KUKA KRL data list: ps_a_ltb_geo_x01.dat

&ACCESS RVO1
&COMMENT Solda Atego LTB
&PARAM DISKPATH = KRC:\R1\Program\OLP
DEFDAT ps_a_ltb_geo_x01
;FOLD EXTERNAL DECLARATIONS;%{PE}%MKUKATPBASIS,%CEXT,%VCOMMON,%P
;FOLD GRIPPERTECH EXT
EXT  H50 (INT  :IN,INT  :IN,INT  :IN,GRP_TYP  :IN )
;ENDFOLD (GRIPPERTECH EXT)
;FOLD SPOTTECH EXT
EXT  USERSPOT (S_COMMAND  :IN,SPOT_TYPE  :IN )
;ENDFOLD (SPOTTECH EXT)
;FOLD BASISTECH EXT;%{PE}%MKUKATPBASIS,%CEXT,%VEXT,%P
EXT  BAS (BAS_COMMAND  :IN,REAL  :IN )
DECL INT SUCCESS
;ENDFOLD (BASISTECH EXT)
;FOLD USER EXT;%{E}%MKUKATPUSER,%CEXT,%VEXT,%P
;Make your modifications here

;ENDFOLD (USER EXT)
;ENDFOLD (EXTERNAL DECLARATIONS)
DECL FDAT Fl005={TOOL_NO 2,BASE_NO 3,IPO_FRAME #BASE,POINT2[] " ",TQ_STATE FALSE}
DECL PDAT PP_OLP2={VEL 100.0,ACC 100.0,APO_DIST 20.0,APO_MODE #CDIS}
DECL E6POS Xl005={X 1312.45898,Y 161.401306,Z 2358.82397,A 138.055695,B 49.2517204,C -31.9309597,S 2,T 10,E1 0.0,E2 0.0,E3 0.0,E4 0.0,E5 0.0,E6 0.0}
DECL FDAT Fl010={TOOL_NO 2,BASE_NO 3,IPO_FRAME #BASE,POINT2[] " "}
DECL PDAT PP_OLP3={VEL 100.0,ACC 100.0,APO_DIST 20.0,APO_MODE #CDIS}
DECL E6POS Xl010={X 1099.32495,Y 478.981415,Z 1743.81201,A 120.314499,B 19.6099892,C -13.0668297,S 2,T 10,E1 0.0,E2 0.0,E3 0.0,E4 0.0,E5 0.0,E6 0.0}
DECL FDAT Fl015={TOOL_NO 2,BASE_NO 3,IPO_FRAME #BASE,POINT2[] " ",TQ_STATE FALSE}
DECL E6POS Xl015={X 661.974487,Y 862.0224,Z 1485.94897,A 120.333702,B 9.80480957,C -0.70352149,S 2,T 10,E1 0.0,E2 0.0,E3 0.0,E4 0.0,E5 0.0,E6 0.0}
DECL FDAT Fl020={TOOL_NO 2,BASE_NO 3,IPO_FRAME #BASE,POINT2[] " ",TQ_STATE FALSE}
DECL PDAT PP_OLP4={VEL 100.0,ACC 100.0,APO_DIST 1.0,APO_MODE #CDIS}
DECL E6POS Xl020={X 658.155701,Y 906.481018,Z 1479.59802,A 120.333801,B 9.80491829,C -0.703368127,S 2,T 10,E1 0.0,E2 0.0,E3 0.0,E4 0.0,E5 0.0,E6 0.0}
DECL FDAT FSWP_60_9850={TOOL_NO 2,BASE_NO 3,IPO_FRAME #BASE,POINT2[] " ",TQ_STATE FALSE}
DECL E6POS XSWP_60_9850={X 650.992371,Y 922.430725,Z 1484.68604,A 120.333,B 9.8059864,C -0.703050911,S 2,T 10,E1 0.0,E2 0.0,E3 0.0,E4 0.0,E5 0.0,E6 0.0}
DECL LDAT LL_OLP2={VEL 2.0,ACC 100.0,APO_DIST 0.0,APO_FAC 0.0,ORI_TYP #VAR,CIRC_TYP #BASE,JERK_FAC 50.0}
DECL FDAT Fl025={TOOL_NO 2,BASE_NO 3,IPO_FRAME #BASE,POINT2[] " ",TQ_STATE FALSE}
DECL PDAT PP_OLP5={VEL 100.0,ACC 100.0,APO_DIST 1.0,APO_MODE #CDIS}
DECL E6POS Xl025={X 673.995117,Y 879.40979,Z 1485.01794,A 120.333801,B 9.80493546,C -0.703359783,S 2,T 10,E1 0.0,E2 0.0,E3 0.0,E4 0.0,E5 0.0,E6 0.0}
DECL FDAT Fl030={TOOL_NO 2,BASE_NO 3,IPO_FRAME #BASE,POINT2[] " "}
DECL PDAT PP_OLP6={VEL 100.0,ACC 100.0,APO_DIST 20.0,APO_MODE #CDIS}
DECL E6POS Xl030={X 679.488281,Y 831.263184,Z 1526.35303,A 120.333801,B 9.80495071,C -0.703492999,S 2,T 10,E1 0.0,E2 0.0,E3 0.0,E4 0.0,E5 0.0,E6 0.0}
DECL FDAT Fl075={TOOL_NO 2,BASE_NO 3,IPO_FRAME #BASE,POINT2[] " "}
DECL PDAT PP_OLP12={VEL 100.0,ACC 100.0,APO_DIST 10.0,APO_MODE #CDIS}
DECL E6POS Xl075={X 1053.93103,Y 888.187012,Z 1501.89294,A 110.206001,B 7.66410017,C 0.278800011,S 2,T 10}
DECL FDAT Fl080={TOOL_NO 2,BASE_NO 3,IPO_FRAME #BASE,POINT2[] " ",TQ_STATE FALSE}
DECL PDAT PP_OLP13={VEL 100.0,ACC 100.0,APO_DIST 1.0,APO_MODE #CDIS}
DECL E6POS Xl080={X 1042.37305,Y 937.541321,Z 1495.12097,A 110.206001,B 7.66410017,C 0.278799713,S 2,T 10,E1 0.0,E2 0.0,E3 0.0,E4 0.0,E5 0.0,E6 0.0}
DECL FDAT FSWP_60_9830={TOOL_NO 2,BASE_NO 3,IPO_FRAME #BASE,POINT2[] " ",TQ_STATE FALSE}
DECL E6POS XSWP_60_9830={X 1047.45996,Y 935.341187,Z 1503.255,A 105.468498,B 7.6633358,C -0.35240531,S 2,T 10,E1 0.0,E2 0.0,E3 0.0,E4 0.0,E5 0.0,E6 0.0}
DECL LDAT LL_OLP7={VEL 2.0,ACC 100.0,APO_DIST 0.0,APO_FAC 0.0,ORI_TYP #VAR,CIRC_TYP #BASE,JERK_FAC 50.0}
DECL FDAT Fl085={TOOL_NO 2,BASE_NO 3,IPO_FRAME #BASE,POINT2[] " ",TQ_STATE FALSE}
DECL PDAT PP_OLP14={VEL 100.0,ACC 100.0,APO_DIST 10.0,APO_MODE #CDIS}
DECL E6POS Xl085={X 1047.91394,Y 934.013428,Z 1492.54199,A 110.206001,B 7.66410017,C 0.278799713,S 2,T 10,E1 0.0,E2 0.0,E3 0.0,E4 0.0,E5 0.0,E6 0.0}
DECL FDAT Fl090={TOOL_NO 2,BASE_NO 3,IPO_FRAME #BASE,POINT2[] " "}
DECL PDAT PP_OLP15={VEL 100.0,ACC 100.0,APO_DIST 20.0,APO_MODE #CDIS}
DECL E6POS Xl090={X 1054.13501,Y 877.552979,Z 1496.93701,A 110.206001,B 7.66410017,C 0.278800011,S 2,T 10}
DECL FDAT Fl095={TOOL_NO 2,BASE_NO 3,IPO_FRAME #BASE,POINT2[] " "}
DECL PDAT PP_OLP16={VEL 100.0,ACC 100.0,APO_DIST 20.0,APO_MODE #CDIS}
DECL E6POS Xl095={X 1235.46899,Y 833.687683,Z 1509.99805,A 95.0815277,B 7.10638905,C -1.278669,S 2,T 10,E1 0.0,E2 0.0,E3 0.0,E4 0.0,E5 0.0,E6 0.0}
DECL FDAT Fl100={TOOL_NO 2,BASE_NO 3,IPO_FRAME #BASE,POINT2[] " "}
DECL PDAT PP_OLP17={VEL 100.0,ACC 100.0,APO_DIST 1.0,APO_MODE #CDIS}
DECL E6POS Xl100={X 1220.69995,Y 941.12323,Z 1501.41797,A 95.0815964,B 7.10640001,C -0.278800011,S 2,T 10,E1 0.0,E2 0.0,E3 0.0,E4 0.0,E5 0.0,E6 0.0}
DECL FDAT FSWP_60_9820={TOOL_NO 2,BASE_NO 3,IPO_FRAME #BASE,POINT2[] " ",TQ_STATE FALSE}
DECL E6POS XSWP_60_9820={X 1228.35999,Y 938.071594,Z 1507.35901,A 95.0815964,B 7.10639477,C -0.278758287,S 2,T 10,E1 0.0,E2 0.0,E3 0.0,E4 0.0,E5 0.0,E6 0.0}
DECL LDAT LL_OLP8={VEL 2.0,ACC 100.0,APO_DIST 0.0,APO_FAC 0.0,ORI_TYP #VAR,CIRC_TYP #BASE,JERK_FAC 50.0}
DECL FDAT Fl105={TOOL_NO 2,BASE_NO 3,IPO_FRAME #BASE,POINT2[] " ",TQ_STATE FALSE}
DECL PDAT PP_OLP18={VEL 100.0,ACC 100.0,APO_DIST 5.0,APO_MODE #CDIS}
DECL E6POS Xl105={X 1221.16797,Y 935.86438,Z 1502.07605,A 95.0815964,B 7.10640001,C -0.278800011,S 2,T 10,E1 0.0,E2 0.0,E3 0.0,E4 0.0,E5 0.0,E6 0.0}
DECL FDAT Fl110={TOOL_NO 2,BASE_NO 3,IPO_FRAME #BASE,POINT2[] " "}
DECL PDAT PP_OLP19={VEL 100.0,ACC 100.0,APO_DIST 20.0,APO_MODE #CDIS}
DECL E6POS Xl110={X 1240.21802,Y 780.291016,Z 1516.68005,A 95.0814972,B 7.10640001,C -1.27869999,S 2,T 10}
DECL FDAT Fl115={TOOL_NO 2,BASE_NO 3,IPO_FRAME #BASE,POINT2[] " "}
DECL PDAT PP_OLP20={VEL 100.0,ACC 100.0,APO_DIST 20.0,APO_MODE #CDIS}
DECL E6POS Xl115={X 1330.44897,Y 420.916992,Z 1021.96503,A 41.7639008,B 75.9056015,C 134.514694,S 2,T 10}
DECL FDAT Fl120={TOOL_NO 2,BASE_NO 3,IPO_FRAME #BASE,POINT2[] " "}
DECL PDAT PP_OLP21={VEL 100.0,ACC 100.0,APO_DIST 10.0,APO_MODE #CDIS}
DECL E6POS Xl120={X 1430.45703,Y 920.916016,Z 371.963013,A 69.623497,B 58.540699,C 160.565796,S 2,T 8}
DECL FDAT Fl125={TOOL_NO 2,BASE_NO 3,IPO_FRAME #BASE,POINT2[] " "}
DECL PDAT PP_OLP22={VEL 100.0,ACC 100.0,APO_DIST 1.0,APO_MODE #CDIS}
DECL E6POS Xl125={X 1430.50403,Y 1010.90399,Z 366.421509,A 69.6233978,B 58.540699,C 160.565704,S 2,T 8,E1 0.0,E2 0.0,E3 0.0,E4 0.0,E5 0.0,E6 0.0}
DECL FDAT Fl130={TOOL_NO 2,BASE_NO 3,IPO_FRAME #BASE,POINT2[] " ",TQ_STATE FALSE}
DECL E6POS Xl130={X 1432.80505,Y 1017.59302,Z 344.019592,A 60.8482018,B 67.7460022,C 152.708603,S 2,T 8,E1 0.0,E2 0.0,E3 0.0,E4 0.0,E5 0.0,E6 0.0}
DECL LDAT LL_OLP9={VEL 1.0,ACC 100.0,APO_DIST 1.0,APO_FAC 0.0,ORI_TYP #VAR,CIRC_TYP #BASE,JERK_FAC 50.0}
DECL FDAT Fl135={TOOL_NO 2,BASE_NO 3,IPO_FRAME #BASE,POINT2[] " "}
DECL E6POS Xl135={X 1404.30798,Y 1011.31897,Z 333.189606,A 176.413498,B 85.4335403,C -90.0502014,S 2,T 9,E1 0.0,E2 0.0,E3 0.0,E4 0.0,E5 0.0,E6 0.0}
DECL LDAT LL_OLP10={VEL 1.0,ACC 100.0,APO_DIST 1.0,APO_FAC 0.0,ORI_TYP #VAR,CIRC_TYP #BASE,JERK_FAC 50.0}
DECL FDAT FSWP_60_9556={TOOL_NO 2,BASE_NO 3,IPO_FRAME #BASE,POINT2[] " ",TQ_STATE FALSE}
DECL E6POS XSWP_60_9556={X 1399.95203,Y 1005.73297,Z 339.989105,A 176.371597,B 82.4862366,C -89.9990616,S 2,T 41,E1 0.0,E2 0.0,E3 0.0,E4 0.0,E5 0.0,E6 0.0}
DECL LDAT LL_OLP11={VEL 2.0,ACC 100.0,APO_DIST 0.0,APO_FAC 0.0,ORI_TYP #VAR,CIRC_TYP #BASE,JERK_FAC 50.0}
DECL FDAT FSWP_60_9568={TOOL_NO 2,BASE_NO 3,IPO_FRAME #BASE,POINT2[] " ",TQ_STATE FALSE}
DECL E6POS XSWP_60_9568={X 1572.35706,Y 996.624878,Z 306.298309,A -3.66327906,B 52.9997711,C 89.9598618,S 2,T 9,E1 0.0,E2 0.0,E3 0.0,E4 0.0,E5 0.0,E6 0.0}
DECL LDAT LL_OLP14={VEL 2.0,ACC 100.0,APO_DIST 0.0,APO_FAC 0.0,ORI_TYP #VAR,CIRC_TYP #BASE,JERK_FAC 50.0}
DECL FDAT Fl150={TOOL_NO 2,BASE_NO 3,IPO_FRAME #BASE,POINT2[] " ",TQ_STATE FALSE}
DECL E6POS Xl150={X 1501.948,Y 1015.54901,Z 314.006989,A 6.11479998,B 59.6772995,C 97.5519028,S 2,T 9,E1 0.0,E2 0.0,E3 0.0,E4 0.0,E5 0.0,E6 0.0}
DECL LDAT LL_OLP15={VEL 1.0,ACC 100.0,APO_DIST 5.0,APO_FAC 0.0,ORI_TYP #VAR,CIRC_TYP #BASE,JERK_FAC 50.0}
DECL FDAT Fl155={TOOL_NO 2,BASE_NO 3,IPO_FRAME #BASE,POINT2[] " "}
DECL E6POS Xl155={X 1430.505,Y 1010.64301,Z 363.86969,A 69.623497,B 58.540699,C 160.565704,S 2,T 8,E1 0.0,E2 0.0,E3 0.0,E4 0.0,E5 0.0,E6 0.0}
DECL LDAT LL_OLP16={VEL 1.0,ACC 100.0,APO_DIST 2.0,APO_FAC 0.0,ORI_TYP #VAR,CIRC_TYP #BASE,JERK_FAC 50.0}
DECL FDAT Fl160={TOOL_NO 2,BASE_NO 3,IPO_FRAME #BASE,POINT2[] " ",TQ_STATE FALSE}
DECL PDAT PP_OLP23={VEL 100.0,ACC 100.0,APO_DIST 10.0,APO_MODE #CDIS}
DECL E6POS Xl160={X 1430.45496,Y 920.916016,Z 371.963013,A 69.623497,B 58.540699,C 160.565704,S 2,T 8}
DECL FDAT Fl165={TOOL_NO 2,BASE_NO 3,IPO_FRAME #BASE,POINT2[] " "}
DECL PDAT PP_OLP24={VEL 100.0,ACC 100.0,APO_DIST 20.0,APO_MODE #CDIS}
DECL E6POS Xl165={X 2150.21997,Y 916.004028,Z 296.890991,A 90.0,B 50.0000992,C -90.0,S 2,T 41}
DECL FDAT Fl170={TOOL_NO 2,BASE_NO 3,IPO_FRAME #BASE,POINT2[] " ",TQ_STATE FALSE}
DECL E6POS Xl170={X 2210.22095,Y 936.007019,Z 296.891998,A 76.0688019,B 44.0681992,C -100.668999,S 2,T 41}
DECL LDAT LL_OLP17={VEL 1.0,ACC 100.0,APO_DIST 5.0,APO_FAC 0.0,ORI_TYP #VAR,CIRC_TYP #BASE,JERK_FAC 50.0}
DECL FDAT Fl175={TOOL_NO 2,BASE_NO 3,IPO_FRAME #BASE,POINT2[] " "}
DECL E6POS Xl175={X 2210.23511,Y 950.996521,Z 278.219299,A 90.0002594,B 50.0004005,C -89.9997406,S 2,T 41,E1 0.0,E2 0.0,E3 0.0,E4 0.0,E5 0.0,E6 0.0}
DECL LDAT LL_OLP18={VEL 1.0,ACC 100.0,APO_DIST 1.0,APO_FAC 0.0,ORI_TYP #VAR,CIRC_TYP #BASE,JERK_FAC 50.0}
DECL FDAT FSWP_60_9456={TOOL_NO 2,BASE_NO 3,IPO_FRAME #BASE,POINT2[] " ",TQ_STATE FALSE}
DECL E6POS XSWP_60_9456={X 2205.08203,Y 972.187317,Z 273.574799,A 98.7543564,B 49.6729088,C -83.3060226,S 2,T 41,E1 0.0,E2 0.0,E3 0.0,E4 0.0,E5 0.0,E6 0.0}
DECL LDAT LL_OLP19={VEL 2.0,ACC 100.0,APO_DIST 0.0,APO_FAC 0.0,ORI_TYP #VAR,CIRC_TYP #BASE,JERK_FAC 50.0}
DECL FDAT Fl180={TOOL_NO 2,BASE_NO 3,IPO_FRAME #BASE,POINT2[] " ",TQ_STATE FALSE}
DECL E6POS Xl180={X 2208.22998,Y 950.996582,Z 277.63559,A 90.000267,B 50.0004005,C -89.9997406,S 2,T 41,E1 0.0,E2 0.0,E3 0.0,E4 0.0,E5 0.0,E6 0.0}
DECL LDAT LL_OLP20={VEL 1.0,ACC 100.0,APO_DIST 5.0,APO_FAC 0.0,ORI_TYP #VAR,CIRC_TYP #BASE,JERK_FAC 50.0}
DECL FDAT Fl185={TOOL_NO 2,BASE_NO 3,IPO_FRAME #BASE,POINT2[] " "}
DECL E6POS Xl185={X 2214.52905,Y 863.063171,Z 284.3349,A 90.0,B 70.0,C -90.0,S 2,T 41,E1 0.0,E2 0.0,E3 0.0,E4 0.0,E5 0.0,E6 0.0}
DECL LDAT LL_OLP21={VEL 1.0,ACC 100.0,APO_DIST 5.0,APO_FAC 0.0,ORI_TYP #VAR,CIRC_TYP #BASE,JERK_FAC 50.0}
DECL FDAT FSWP_60_9446={TOOL_NO 2,BASE_NO 3,IPO_FRAME #BASE,POINT2[] " ",TQ_STATE FALSE}
DECL E6POS XSWP_60_9446={X 2208.25293,Y 831.700378,Z 279.504791,A 90.0002136,B 70.0000229,C -89.9997864,S 2,T 41,E1 0.0,E2 0.0,E3 0.0,E4 0.0,E5 0.0,E6 0.0}
DECL LDAT LL_OLP22={VEL 2.0,ACC 100.0,APO_DIST 0.0,APO_FAC 0.0,ORI_TYP #VAR,CIRC_TYP #BASE,JERK_FAC 50.0}
DECL FDAT Fl195={TOOL_NO 2,BASE_NO 3,IPO_FRAME #BASE,POINT2[] " "}
DECL E6POS Xl195={X 2205.21704,Y 709.570007,Z 304.463013,A 90.0,B 70.0,C -90.0,S 2,T 41}
DECL LDAT LL_OLP24={VEL 1.0,ACC 100.0,APO_DIST 5.0,APO_FAC 0.0,ORI_TYP #VAR,CIRC_TYP #BASE,JERK_FAC 50.0}
DECL FDAT Fl200={TOOL_NO 2,BASE_NO 3,IPO_FRAME #BASE,POINT2[] " "}
DECL E6POS Xl200={X 2210.23608,Y 593.166016,Z 330.933594,A 78.6753998,B 84.9012985,C -101.280998,S 2,T 9,E1 0.0,E2 0.0,E3 0.0,E4 0.0,E5 0.0,E6 0.0}
DECL LDAT LL_OLP25={VEL 1.0,ACC 100.0,APO_DIST 5.0,APO_FAC 0.0,ORI_TYP #VAR,CIRC_TYP #BASE,JERK_FAC 50.0}
DECL FDAT FSWP_60_9436={TOOL_NO 2,BASE_NO 3,IPO_FRAME #BASE,POINT2[] " ",TQ_STATE FALSE}
DECL E6POS XSWP_60_9436={X 2207.03711,Y 588.41748,Z 325.153595,A 136.424805,B 82.7309265,C -43.8064194,S 2,T 9,E1 0.0,E2 0.0,E3 0.0,E4 0.0,E5 0.0,E6 0.0}
DECL LDAT LL_OLP26={VEL 2.0,ACC 100.0,APO_DIST 0.0,APO_FAC 0.0,ORI_TYP #VAR,CIRC_TYP #BASE,JERK_FAC 50.0}
DECL FDAT Fl205={TOOL_NO 2,BASE_NO 3,IPO_FRAME #BASE,POINT2[] " ",TQ_STATE FALSE}
DECL E6POS Xl205={X 2210.21411,Y 578.169006,Z 340.212006,A 90.0,B 85.0,C -89.9999008,S 2,T 9}
DECL LDAT LL_OLP27={VEL 1.0,ACC 100.0,APO_DIST 5.0,APO_FAC 0.0,ORI_TYP #VAR,CIRC_TYP #BASE,JERK_FAC 50.0}
DECL FDAT Fl210={TOOL_NO 2,BASE_NO 3,IPO_FRAME #BASE,POINT2[] " "}
DECL E6POS Xl210={X 2205.22095,Y 478.169006,Z 460.212006,A 90.0,B 85.0,C -90.0,S 2,T 9}
DECL LDAT LL_OLP28={VEL 1.0,ACC 100.0,APO_DIST 50.0,APO_FAC 0.0,ORI_TYP #VAR,CIRC_TYP #BASE,JERK_FAC 50.0}
DECL FDAT Fl215={TOOL_NO 2,BASE_NO 3,IPO_FRAME #BASE,POINT2[] " "}
DECL E6POS Xl215={X 2212.68994,Y 350.626801,Z 477.752014,A -58.9805984,B 84.1710968,C 120.888397,S 2,T 9,E1 0.0,E2 0.0,E3 0.0,E4 0.0,E5 0.0,E6 0.0}
DECL LDAT LL_OLP29={VEL 1.0,ACC 100.0,APO_DIST 1.0,APO_FAC 0.0,ORI_TYP #VAR,CIRC_TYP #BASE,JERK_FAC 50.0}
DECL FDAT FSWP_60_9418={TOOL_NO 2,BASE_NO 3,IPO_FRAME #BASE,POINT2[] " ",TQ_STATE FALSE}
DECL E6POS XSWP_60_9418={X 2208.3291,Y 339.465393,Z 466.934204,A -153.915298,B 84.7714386,C 26.7148399,S 2,T 9,E1 0.0,E2 0.0,E3 0.0,E4 0.0,E5 0.0,E6 0.0}
DECL LDAT LL_OLP30={VEL 2.0,ACC 100.0,APO_DIST 0.0,APO_FAC 0.0,ORI_TYP #VAR,CIRC_TYP #BASE,JERK_FAC 50.0}
DECL FDAT Fl220={TOOL_NO 2,BASE_NO 3,IPO_FRAME #BASE,POINT2[] " ",TQ_STATE FALSE}
DECL E6POS Xl220={X 2210.22192,Y 329.837006,Z 477.765991,A -90.0002975,B 85.0000992,C 89.9997025,S 2,T 9}
DECL LDAT LL_OLP31={VEL 1.0,ACC 100.0,APO_DIST 5.0,APO_FAC 0.0,ORI_TYP #VAR,CIRC_TYP #BASE,JERK_FAC 50.0}
DECL FDAT Fl225={TOOL_NO 2,BASE_NO 3,IPO_FRAME #BASE,POINT2[] " "}
DECL E6POS Xl225={X 2205.26099,Y 224.826096,Z 516.190002,A -26.3003006,B 78.8312988,C 153.256699,S 2,T 9,E1 0.0,E2 0.0,E3 0.0,E4 0.0,E5 0.0,E6 0.0}
DECL LDAT LL_OLP32={VEL 1.0,ACC 100.0,APO_DIST 10.0,APO_FAC 0.0,ORI_TYP #VAR,CIRC_TYP #BASE,JERK_FAC 50.0}
DECL FDAT Fl230={TOOL_NO 2,BASE_NO 3,IPO_FRAME #BASE,POINT2[] " "}
DECL E6POS Xl230={X 2209.88208,Y 85.7576523,Z 494.679993,A -78.4449997,B 69.6200027,C 100.849403,S 2,T 9,E1 0.0,E2 0.0,E3 0.0,E4 0.0,E5 0.0,E6 0.0}
DECL LDAT LL_OLP33={VEL 1.0,ACC 100.0,APO_DIST 5.0,APO_FAC 0.0,ORI_TYP #VAR,CIRC_TYP #BASE,JERK_FAC 50.0}
DECL FDAT FSWP_60_9402={TOOL_NO 2,BASE_NO 3,IPO_FRAME #BASE,POINT2[] " ",TQ_STATE FALSE}
DECL E6POS XSWP_60_9402={X 2206.31909,Y 39.0832901,Z 481.429993,A -103.966202,B 69.3978119,C 76.3905563,S 2,T 9,E1 0.0,E2 0.0,E3 0.0,E4 0.0,E5 0.0,E6 0.0}
DECL LDAT LL_OLP34={VEL 2.0,ACC 100.0,APO_DIST 0.0,APO_FAC 0.0,ORI_TYP #VAR,CIRC_TYP #BASE,JERK_FAC 50.0}
DECL FDAT Fl235={TOOL_NO 2,BASE_NO 3,IPO_FRAME #BASE,POINT2[] " ",TQ_STATE FALSE}
DECL E6POS Xl235={X 2209.8811,Y 85.7577896,Z 502.071899,A -78.4450607,B 69.6199722,C 100.849297,S 2,T 9,E1 0.0,E2 0.0,E3 0.0,E4 0.0,E5 0.0,E6 0.0}
DECL LDAT LL_OLP35={VEL 1.0,ACC 100.0,APO_DIST 10.0,APO_FAC 0.0,ORI_TYP #VAR,CIRC_TYP #BASE,JERK_FAC 50.0}
DECL FDAT Fl240={TOOL_NO 2,BASE_NO 3,IPO_FRAME #BASE,POINT2[] " "}
DECL E6POS Xl240={X 2125.229,Y 51.7761002,Z 518.945007,A -48.5031395,B 67.3752823,C 118.888,S 2,T 9,E1 0.0,E2 0.0,E3 0.0,E4 0.0,E5 0.0,E6 0.0}
DECL LDAT LL_OLP36={VEL 1.0,ACC 100.0,APO_DIST 20.0,APO_FAC 0.0,ORI_TYP #VAR,CIRC_TYP #BASE,JERK_FAC 50.0}
DECL FDAT Fl245={TOOL_NO 2,BASE_NO 3,IPO_FRAME #BASE,POINT2[] " "}
DECL E6POS Xl245={X 2125.2229,Y -51.7659988,Z 501.994995,A 48.5036011,B 67.3753967,C -118.887802,S 2,T 40}
DECL LDAT LL_OLP37={VEL 1.0,ACC 100.0,APO_DIST 101.0,APO_FAC 0.0,ORI_TYP #VAR,CIRC_TYP #BASE,JERK_FAC 50.0}
DECL FDAT Fl250={TOOL_NO 2,BASE_NO 3,IPO_FRAME #BASE,POINT2[] " "}
DECL E6POS Xl250={X 2210.22192,Y -87.8785324,Z 501.994995,A 48.5036011,B 67.3753967,C -118.887802,S 2,T 40,E1 0.0,E2 0.0,E3 0.0,E4 0.0,E5 0.0,E6 0.0}
DECL LDAT LL_OLP38={VEL 1.0,ACC 100.0,APO_DIST 5.0,APO_FAC 0.0,ORI_TYP #VAR,CIRC_TYP #BASE,JERK_FAC 50.0}
DECL FDAT Fl255={TOOL_NO 2,BASE_NO 3,IPO_FRAME #BASE,POINT2[] " "}
DECL E6POS Xl255={X 2213.58691,Y -83.7550735,Z 486.702515,A 75.2710037,B 70.2698975,C -93.8613968,S 2,T 40,E1 0.0,E2 0.0,E3 0.0,E4 0.0,E5 0.0,E6 0.0}
DECL LDAT LL_OLP39={VEL 1.0,ACC 100.0,APO_DIST 2.0,APO_FAC 0.0,ORI_TYP #VAR,CIRC_TYP #BASE,JERK_FAC 50.0}
DECL FDAT FSWP_60_9401={TOOL_NO 2,BASE_NO 3,IPO_FRAME #BASE,POINT2[] " ",TQ_STATE FALSE}
DECL E6POS XSWP_60_9401={X 2209.38892,Y -45.844059,Z 480.638794,A 102.350197,B 69.5346603,C -77.8060226,S 2,T 40,E1 0.0,E2 0.0,E3 0.0,E4 0.0,E5 0.0,E6 0.0}
DECL LDAT LL_OLP40={VEL 2.0,ACC 100.0,APO_DIST 0.0,APO_FAC 0.0,ORI_TYP #VAR,CIRC_TYP #BASE,JERK_FAC 50.0}
DECL FDAT Fl260={TOOL_NO 2,BASE_NO 3,IPO_FRAME #BASE,POINT2[] " ",TQ_STATE FALSE}
DECL E6POS Xl260={X 2210.19409,Y -226.362305,Z 515.516724,A 26.3024998,B 78.8311005,C -153.259796,S 2,T 8,E1 0.0,E2 0.0,E3 0.0,E4 0.0,E5 0.0,E6 0.0}
DECL LDAT LL_OLP41={VEL 1.0,ACC 100.0,APO_DIST 5.0,APO_FAC 0.0,ORI_TYP #VAR,CIRC_TYP #BASE,JERK_FAC 50.0}
DECL FDAT Fl265={TOOL_NO 2,BASE_NO 3,IPO_FRAME #BASE,POINT2[] " "}
DECL E6POS Xl265={X 2211.18408,Y -349.819397,Z 475.749908,A 89.4250107,B 88.7149429,C -90.5897598,S 2,T 8,E1 0.0,E2 0.0,E3 0.0,E4 0.0,E5 0.0,E6 0.0}
DECL LDAT LL_OLP42={VEL 1.0,ACC 100.0,APO_DIST 5.0,APO_FAC 0.0,ORI_TYP #VAR,CIRC_TYP #BASE,JERK_FAC 50.0}
DECL FDAT FSWP_60_9417={TOOL_NO 2,BASE_NO 3,IPO_FRAME #BASE,POINT2[] " ",TQ_STATE FALSE}
DECL E6POS XSWP_60_9417={X 2209.16406,Y -352.611694,Z 465.538605,A 165.204895,B 84.2824936,C -14.6828499,S 2,T 8,E1 0.0,E2 0.0,E3 0.0,E4 0.0,E5 0.0,E6 0.0}
DECL LDAT LL_OLP43={VEL 2.0,ACC 100.0,APO_DIST 0.0,APO_FAC 0.0,ORI_TYP #VAR,CIRC_TYP #BASE,JERK_FAC 50.0}
DECL FDAT Fl270={TOOL_NO 2,BASE_NO 3,IPO_FRAME #BASE,POINT2[] " ",TQ_STATE FALSE}
DECL E6POS Xl270={X 2205.22095,Y -478.169006,Z 460.212006,A -90.0,B 85.0,C 90.0,S 2,T 8}
DECL LDAT LL_OLP44={VEL 1.0,ACC 100.0,APO_DIST 5.0,APO_FAC 0.0,ORI_TYP #VAR,CIRC_TYP #BASE,JERK_FAC 50.0}
DECL FDAT FSWP_60_9435={TOOL_NO 2,BASE_NO 3,IPO_FRAME #BASE,POINT2[] " ",TQ_STATE FALSE}
DECL E6POS XSWP_60_9435={X 2206.49805,Y -596.194885,Z 325.749603,A -126.132797,B 83.7971497,C 53.8362885,S 2,T 8,E1 0.0,E2 0.0,E3 0.0,E4 0.0,E5 0.0,E6 0.0}
DECL LDAT LL_OLP45={VEL 2.0,ACC 100.0,APO_DIST 0.0,APO_FAC 0.0,ORI_TYP #VAR,CIRC_TYP #BASE,JERK_FAC 50.0}
DECL FDAT Fl275={TOOL_NO 2,BASE_NO 3,IPO_FRAME #BASE,POINT2[] " ",TQ_STATE FALSE}
DECL E6POS Xl275={X 2205.21704,Y -709.570007,Z 304.463013,A -90.0,B 70.0,C 90.0,S 2,T 8}
DECL LDAT LL_OLP46={VEL 1.0,ACC 100.0,APO_DIST 5.0,APO_FAC 0.0,ORI_TYP #VAR,CIRC_TYP #BASE,JERK_FAC 50.0}
DECL FDAT FSWP_60_9445={TOOL_NO 2,BASE_NO 3,IPO_FRAME #BASE,POINT2[] " ",TQ_STATE FALSE}
DECL E6POS XSWP_60_9445={X 2207.60107,Y -835.695984,Z 272.809509,A -99.4904099,B 69.7042694,C 80.2663193,S 2,T 8,E1 0.0,E2 0.0,E3 0.0,E4 0.0,E5 0.0,E6 0.0}
DECL LDAT LL_OLP47={VEL 2.0,ACC 100.0,APO_DIST 0.0,APO_FAC 0.0,ORI_TYP #VAR,CIRC_TYP #BASE,JERK_FAC 50.0}
DECL FDAT Fl280={TOOL_NO 2,BASE_NO 3,IPO_FRAME #BASE,POINT2[] " ",TQ_STATE FALSE}
DECL E6POS Xl280={X 2205.229,Y -921.711975,Z 294.875,A -90.0,B 50.0000992,C 90.0,S 2,T 8}
DECL LDAT LL_OLP48={VEL 1.0,ACC 100.0,APO_DIST 5.0,APO_FAC 0.0,ORI_TYP #VAR,CIRC_TYP #BASE,JERK_FAC 50.0}
DECL FDAT FSWP_60_9455={TOOL_NO 2,BASE_NO 3,IPO_FRAME #BASE,POINT2[] " ",TQ_STATE FALSE}
DECL E6POS XSWP_60_9455={X 2203.65405,Y -981.330994,Z 273.67099,A -91.5469894,B 49.9690704,C 87.3450394,S 2,T 8,E1 0.0,E2 0.0,E3 0.0,E4 0.0,E5 0.0,E6 0.0}
DECL LDAT LL_OLP49={VEL 2.0,ACC 100.0,APO_DIST 0.0,APO_FAC 0.0,ORI_TYP #VAR,CIRC_TYP #BASE,JERK_FAC 50.0}
DECL FDAT Fl285={TOOL_NO 2,BASE_NO 3,IPO_FRAME #BASE,POINT2[] " ",TQ_STATE FALSE}
DECL E6POS Xl285={X 2205.26904,Y -951.011414,Z 283.177307,A -90.0000916,B 50.0001907,C 89.9999619,S 2,T 8,E1 0.0,E2 0.0,E3 0.0,E4 0.0,E5 0.0,E6 0.0}
DECL LDAT LL_OLP50={VEL 1.0,ACC 100.0,APO_DIST 2.0,APO_FAC 0.0,ORI_TYP #VAR,CIRC_TYP #BASE,JERK_FAC 50.0}
DECL FDAT Fl290={TOOL_NO 2,BASE_NO 3,IPO_FRAME #BASE,POINT2[] " "}
DECL E6POS Xl290={X 2210.24194,Y -936.011597,Z 302.306213,A -74.660202,B 48.9735985,C 101.692101,S 2,T 8,E1 0.0,E2 0.0,E3 0.0,E4 0.0,E5 0.0,E6 0.0}
DECL LDAT LL_OLP51={VEL 1.0,ACC 100.0,APO_DIST 5.0,APO_FAC 0.0,ORI_TYP #VAR,CIRC_TYP #BASE,JERK_FAC 50.0}
DECL FDAT Fl295={TOOL_NO 2,BASE_NO 3,IPO_FRAME #BASE,POINT2[] " "}
DECL E6POS Xl295={X 2150.30005,Y -916.025818,Z 317.780914,A -89.9999924,B 50.0000992,C 90.0,S 2,T 8,E1 0.0,E2 0.0,E3 0.0,E4 0.0,E5 0.0,E6 0.0}
DECL LDAT LL_OLP52={VEL 1.0,ACC 100.0,APO_DIST 20.0,APO_FAC 0.0,ORI_TYP #VAR,CIRC_TYP #BASE,JERK_FAC 50.0}
DECL FDAT Fl300={TOOL_NO 2,BASE_NO 3,IPO_FRAME #BASE,POINT2[] " ",TQ_STATE FALSE}
DECL PDAT PP_OLP25={VEL 100.0,ACC 100.0,APO_DIST 20.0,APO_MODE #CDIS}
DECL E6POS Xl300={X 1430.48596,Y -920.923828,Z 380.326599,A -69.623497,B 58.5407104,C -160.565704,S 2,T 9,E1 0.0,E2 0.0,E3 0.0,E4 0.0,E5 0.0,E6 0.0}
DECL FDAT Fl305={TOOL_NO 2,BASE_NO 3,IPO_FRAME #BASE,POINT2[] " "}
DECL PDAT PP_OLP26={VEL 100.0,ACC 100.0,APO_DIST 5.0,APO_MODE #CDIS}
DECL E6POS Xl305={X 1430.49695,Y -1010.92603,Z 364.68219,A -69.6234894,B 58.5407104,C -160.565704,S 2,T 9,E1 0.0,E2 0.0,E3 0.0,E4 0.0,E5 0.0,E6 0.0}
DECL FDAT Fl310={TOOL_NO 2,BASE_NO 3,IPO_FRAME #BASE,POINT2[] " ",TQ_STATE FALSE}
DECL E6POS Xl310={X 1504.45801,Y -1015.81799,Z 309.69101,A -6.11479998,B 59.6772995,C -97.5519028,S 2,T 40}
DECL LDAT LL_OLP53={VEL 1.0,ACC 100.0,APO_DIST 2.0,APO_FAC 0.0,ORI_TYP #VAR,CIRC_TYP #BASE,JERK_FAC 50.0}
DECL FDAT Fl315={TOOL_NO 2,BASE_NO 3,IPO_FRAME #BASE,POINT2[] " "}
DECL E6POS Xl315={X 1559.32104,Y -1000.73297,Z 296.967987,A 3.66630006,B 55.0000992,C -89.9583969,S 2,T 40}
DECL LDAT LL_OLP54={VEL 1.0,ACC 100.0,APO_DIST 2.0,APO_FAC 0.0,ORI_TYP #VAR,CIRC_TYP #BASE,JERK_FAC 50.0}
DECL FDAT FSWP_60_9567={TOOL_NO 2,BASE_NO 3,IPO_FRAME #BASE,POINT2[] " ",TQ_STATE FALSE}
DECL E6POS XSWP_60_9567={X 1561.53894,Y -999.303223,Z 297.026215,A 3.66697097,B 55.0008392,C -89.9575882,S 2,T 40,E1 0.0,E2 0.0,E3 0.0,E4 0.0,E5 0.0,E6 0.0}
DECL LDAT LL_OLP55={VEL 2.0,ACC 100.0,APO_DIST 0.0,APO_FAC 0.0,ORI_TYP #VAR,CIRC_TYP #BASE,JERK_FAC 50.0}
DECL FDAT FSWP_60_9555={TOOL_NO 2,BASE_NO 3,IPO_FRAME #BASE,POINT2[] " ",TQ_STATE FALSE}
DECL E6POS XSWP_60_9555={X 1399.047,Y -1007.28302,Z 333.780914,A -176.405594,B 80.0015793,C 89.9643173,S 2,T 8,E1 0.0,E2 0.0,E3 0.0,E4 0.0,E5 0.0,E6 0.0}
DECL LDAT LL_OLP57={VEL 2.0,ACC 100.0,APO_DIST 0.0,APO_FAC 0.0,ORI_TYP #VAR,CIRC_TYP #BASE,JERK_FAC 50.0}
DECL FDAT Fl325={TOOL_NO 2,BASE_NO 3,IPO_FRAME #BASE,POINT2[] " ",TQ_STATE FALSE}
DECL E6POS Xl325={X 1408.64404,Y -1022.89801,Z 347.390106,A -119.316399,B 72.0361023,C 145.7341,S 2,T 8,E1 0.0,E2 0.0,E3 0.0,E4 0.0,E5 0.0,E6 0.0}
DECL LDAT LL_OLP58={VEL 1.0,ACC 100.0,APO_DIST 5.0,APO_FAC 0.0,ORI_TYP #VAR,CIRC_TYP #BASE,JERK_FAC 50.0}
DECL FDAT Fl330={TOOL_NO 2,BASE_NO 3,IPO_FRAME #BASE,POINT2[] " "}
DECL E6POS Xl330={X 1430.49805,Y -1010.927,Z 364.586212,A -69.6234894,B 58.5407104,C -160.565796,S 2,T 9,E1 0.0,E2 0.0,E3 0.0,E4 0.0,E5 0.0,E6 0.0}
DECL LDAT LL_OLP59={VEL 1.0,ACC 100.0,APO_DIST 5.0,APO_FAC 0.0,ORI_TYP #VAR,CIRC_TYP #BASE,JERK_FAC 50.0}
DECL FDAT Fl335={TOOL_NO 2,BASE_NO 3,IPO_FRAME #BASE,POINT2[] " "}
DECL E6POS Xl335={X 1430.45801,Y -920.916016,Z 371.963013,A -41.7638016,B 75.9057007,C -134.514694,S 2,T 40}
DECL LDAT LL_OLP60={VEL 1.0,ACC 100.0,APO_DIST 20.0,APO_FAC 0.0,ORI_TYP #VAR,CIRC_TYP #BASE,JERK_FAC 50.0}
DECL FDAT Fl340={TOOL_NO 2,BASE_NO 3,IPO_FRAME #BASE,POINT2[] " ",TQ_STATE FALSE}
DECL PDAT PP_OLP27={VEL 100.0,ACC 100.0,APO_DIST 50.0,APO_MODE #CDIS}
DECL E6POS Xl340={X 1023.37201,Y 195.498001,Z 1177.24402,A -56.0586014,B 67.5304031,C -3.93070006,S 2,T 10}
DECL FDAT Fl345={TOOL_NO 2,BASE_NO 3,IPO_FRAME #BASE,POINT2[] " "}
DECL PDAT PP_OLP28={VEL 100.0,ACC 100.0,APO_DIST 20.0,APO_MODE #CDIS}
DECL E6POS Xl345={X 1231.26501,Y -831.768921,Z 1504.36499,A -95.0813599,B 7.10645723,C 1.27910495,S 6,T 27,E1 0.0,E2 0.0,E3 0.0,E4 0.0,E5 0.0,E6 0.0}
DECL FDAT Fl350={TOOL_NO 2,BASE_NO 3,IPO_FRAME #BASE,POINT2[] " "}
DECL PDAT PP_OLP29={VEL 100.0,ACC 100.0,APO_DIST 2.0,APO_MODE #CDIS}
DECL E6POS Xl350={X 1229.13696,Y -941.847778,Z 1502.84204,A -95.9412231,B 4.54855013,C -6.22060919,S 6,T 27,E1 0.0,E2 0.0,E3 0.0,E4 0.0,E5 0.0,E6 0.0}
DECL FDAT FSWP_60_9819={TOOL_NO 2,BASE_NO 3,IPO_FRAME #BASE,POINT2[] " ",TQ_STATE FALSE}
DECL E6POS XSWP_60_9819={X 1222.802,Y -950.658203,Z 1506.07397,A -95.8159866,B 4.79627705,C 1.52473104,S 6,T 27,E1 0.0,E2 0.0,E3 0.0,E4 0.0,E5 0.0,E6 0.0}
DECL LDAT LL_OLP61={VEL 2.0,ACC 100.0,APO_DIST 0.0,APO_FAC 0.0,ORI_TYP #VAR,CIRC_TYP #BASE,JERK_FAC 50.0}
DECL FDAT Fl355={TOOL_NO 2,BASE_NO 3,IPO_FRAME #BASE,POINT2[] " ",TQ_STATE FALSE}
DECL PDAT PP_OLP30={VEL 100.0,ACC 100.0,APO_DIST 5.0,APO_MODE #CDIS}
DECL E6POS Xl355={X 1229.13696,Y -941.846985,Z 1502.84094,A -95.9412003,B 4.5486021,C -6.22065115,S 6,T 27,E1 0.0,E2 0.0,E3 0.0,E4 0.0,E5 0.0,E6 0.0}
DECL FDAT Fl360={TOOL_NO 2,BASE_NO 3,IPO_FRAME #BASE,POINT2[] " "}
DECL PDAT PP_OLP31={VEL 100.0,ACC 100.0,APO_DIST 10.0,APO_MODE #CDIS}
DECL E6POS Xl360={X 1245.23401,Y -831.894775,Z 1502.57397,A -95.0814972,B 7.10640001,C 1.27869999,S 6,T 27,E1 0.0,E2 0.0,E3 0.0,E4 0.0,E5 0.0,E6 0.0}
DECL FDAT Fl365={TOOL_NO 2,BASE_NO 3,IPO_FRAME #BASE,POINT2[] " ",TQ_STATE FALSE}
DECL PDAT PP_OLP32={VEL 100.0,ACC 100.0,APO_DIST 10.0,APO_MODE #CDIS}
DECL E6POS Xl365={X 1054.13501,Y -877.552979,Z 1496.93701,A -110.206001,B 7.66410017,C -0.278800011,S 6,T 27}
DECL FDAT Fl370={TOOL_NO 2,BASE_NO 3,IPO_FRAME #BASE,POINT2[] " "}
DECL PDAT PP_OLP33={VEL 100.0,ACC 100.0,APO_DIST 5.0,APO_MODE #CDIS}
DECL E6POS Xl370={X 1041.78296,Y -941.79248,Z 1494.52405,A -110.206001,B 7.66410017,C -0.278800011,S 6,T 27,E1 0.0,E2 0.0,E3 0.0,E4 0.0,E5 0.0,E6 0.0}
DECL FDAT FSWP_60_9829={TOOL_NO 2,BASE_NO 3,IPO_FRAME #BASE,POINT2[] " ",TQ_STATE FALSE}
DECL E6POS XSWP_60_9829={X 1048.76794,Y -952.477783,Z 1499.80103,A -110.206299,B 7.66383219,C -0.278844714,S 6,T 26,E1 0.0,E2 0.0,E3 0.0,E4 0.0,E5 0.0,E6 0.0}
DECL LDAT LL_OLP62={VEL 2.0,ACC 100.0,APO_DIST 0.0,APO_FAC 0.0,ORI_TYP #VAR,CIRC_TYP #BASE,JERK_FAC 50.0}
DECL FDAT Fl375={TOOL_NO 2,BASE_NO 3,IPO_FRAME #BASE,POINT2[] " ",TQ_STATE FALSE}
DECL PDAT PP_OLP34={VEL 100.0,ACC 100.0,APO_DIST 10.0,APO_MODE #CDIS}
DECL E6POS Xl375={X 1064.71106,Y -879.495422,Z 1503.45703,A -110.206001,B 7.66410017,C -0.278800011,S 6,T 27,E1 0.0,E2 0.0,E3 0.0,E4 0.0,E5 0.0,E6 0.0}
DECL FDAT Fl380={TOOL_NO 2,BASE_NO 3,IPO_FRAME #BASE,POINT2[] " "}
DECL PDAT PP_OLP35={VEL 100.0,ACC 100.0,APO_DIST 10.0,APO_MODE #CDIS}
DECL E6POS Xl380={X 1070.62,Y -843.634094,Z 1565.01404,A -110.206001,B 7.66410208,C -0.278800696,S 6,T 27,E1 0.0,E2 0.0,E3 0.0,E4 0.0,E5 0.0,E6 0.0}
DECL FDAT Fl385={TOOL_NO 2,BASE_NO 3,IPO_FRAME #BASE,POINT2[] " "}
DECL PDAT PP_OLP36={VEL 100.0,ACC 100.0,APO_DIST 20.0,APO_MODE #CDIS}
DECL E6POS Xl385={X 910.014587,Y -845.905884,Z 1559.67297,A -110.206001,B 7.66410398,C -0.278801888,S 6,T 27,E1 0.0,E2 0.0,E3 0.0,E4 0.0,E5 0.0,E6 0.0}
DECL FDAT Fl420={TOOL_NO 2,BASE_NO 3,IPO_FRAME #BASE,POINT2[] " "}
DECL PDAT PP_OLP40={VEL 100.0,ACC 100.0,APO_DIST 20.0,APO_MODE #CDIS}
DECL E6POS Xl420={X 660.002075,Y -860.751282,Z 1542.66504,A -120.333801,B 9.80494022,C 0.703443885,S 6,T 58,E1 0.0,E2 0.0,E3 0.0,E4 0.0,E5 0.0,E6 0.0}
DECL FDAT Fl425={TOOL_NO 2,BASE_NO 3,IPO_FRAME #BASE,POINT2[] " ",TQ_STATE FALSE}
DECL PDAT PP_OLP41={VEL 100.0,ACC 100.0,APO_DIST 10.0,APO_MODE #CDIS}
DECL E6POS Xl425={X 646.763,Y -884.752014,Z 1480.66895,A -120.333801,B 9.80490017,C 0.703499973,S 6,T 58}
DECL FDAT Fl430={TOOL_NO 2,BASE_NO 3,IPO_FRAME #BASE,POINT2[] " "}
DECL PDAT PP_OLP42={VEL 100.0,ACC 100.0,APO_DIST 2.0,APO_MODE #CDIS}
DECL E6POS Xl430={X 632.411377,Y -939.182617,Z 1471.48401,A -120.333801,B 9.80489922,C 0.703500926,S 6,T 58,E1 0.0,E2 0.0,E3 0.0,E4 0.0,E5 0.0,E6 0.0}
DECL FDAT FSWP_60_9849={TOOL_NO 2,BASE_NO 3,IPO_FRAME #BASE,POINT2[] " ",TQ_STATE FALSE}
DECL E6POS XSWP_60_9849={X 648.606018,Y -944.173279,Z 1474.62,A -110.055496,B 9.46926117,C 2.36206508,S 6,T 58,E1 0.0,E2 0.0,E3 0.0,E4 0.0,E5 0.0,E6 0.0}
DECL LDAT LL_OLP67={VEL 2.0,ACC 100.0,APO_DIST 0.0,APO_FAC 0.0,ORI_TYP #VAR,CIRC_TYP #BASE,JERK_FAC 50.0}
DECL FDAT Fl435={TOOL_NO 2,BASE_NO 3,IPO_FRAME #BASE,POINT2[] " ",TQ_STATE FALSE}
DECL E6POS Xl435={X 632.411377,Y -939.182617,Z 1471.48401,A -120.333801,B 9.80489922,C 0.703500926,S 6,T 58,E1 0.0,E2 0.0,E3 0.0,E4 0.0,E5 0.0,E6 0.0}
DECL FDAT Fl440={TOOL_NO 2,BASE_NO 3,IPO_FRAME #BASE,POINT2[] " "}
DECL PDAT PP_OLP44={VEL 100.0,ACC 100.0,APO_DIST 10.0,APO_MODE #CDIS}
DECL E6POS Xl440={X 646.763977,Y -884.752014,Z 1480.66895,A -120.333801,B 9.80490017,C 0.703499973,S 6,T 58}
DECL FDAT Fl445={TOOL_NO 2,BASE_NO 3,IPO_FRAME #BASE,POINT2[] " ",TQ_STATE FALSE}
DECL E6POS Xl445={X 903.630981,Y -565.390015,Z 1544.61304,A -115.101402,B 14.6844997,C 2.03340006,S 6,T 27}
DECL LDAT LL_OLP68={VEL 1.0,ACC 100.0,APO_DIST 50.0,APO_FAC 0.0,ORI_TYP #VAR,CIRC_TYP #BASE,JERK_FAC 50.0}
DECL FDAT Fl450={TOOL_NO 2,BASE_NO 3,IPO_FRAME #BASE,POINT2[] " ",TQ_STATE FALSE}
DECL PDAT PP_OLP45={VEL 100.0,ACC 100.0,APO_DIST 50.0,APO_MODE #CDIS}
DECL E6POS Xl450={X 1399.95703,Y -542.234924,Z 2580.37402,A -75.9914017,B 22.5326004,C -25.0158005,S 6,T 27,E1 0.0,E2 0.0,E3 0.0,E4 0.0,E5 0.0,E6 0.0}
DECL BASIS_SUGG_T LAST_BASIS={POINT1[] "P0                      ",POINT2[] "P0                      ",CP_PARAMS[] "CPDAT0                  ",PTP_PARAMS[] "PDAT0                   ",CONT[] "                        ",CP_VEL[] "2.0                     ",PTP_VEL[] " 100                    ",SYNC_PARAMS[] "SYNCDAT                 ",SPL_NAME[] "S0                      "}
DECL PDAT PP_OLP47={VEL 100.0,ACC 100.0,APO_DIST 50.0,APO_MODE #CDIS}
DECL E6POS Xl006={X 1052.75195,Y 58.7190018,Z 2073.41504,A -29.1716995,B 74.7963028,C -24.9258003,S 2,T 3}
DECL FDAT Fl006={TOOL_NO 2,BASE_NO 3,IPO_FRAME #BASE,POINT2[] " ",TQ_STATE FALSE}
DECL PDAT PP_OLP48={VEL 100.0,ACC 100.0,APO_DIST 0.0}
DECL E6POS Xl011={X 788.399475,Y 515.901306,Z 807.937988,A -165.150803,B 79.6066818,C -105.500198,S 2,T 8,E1 0.0,E2 0.0,E3 0.0,E4 0.0,E5 0.0,E6 0.0}
DECL FDAT Fl011={TOOL_NO 2,BASE_NO 3,IPO_FRAME #BASE,POINT2[] " ",TQ_STATE FALSE}
DECL LDAT LL_OLP69={VEL 2.0,ACC 100.0,APO_DIST 50.0,APO_FAC 0.0,ORI_TYP #VAR,CIRC_TYP #BASE,JERK_FAC 50.0}
DECL E6POS Xl016={X 293.170685,Y 908.471497,Z -4.25657701,A -179.468506,B 64.3328323,C -98.5837173,S 2,T 41,E1 0.0,E2 0.0,E3 0.0,E4 0.0,E5 0.0,E6 0.0}
DECL FDAT Fl016={TOOL_NO 2,BASE_NO 3,IPO_FRAME #BASE,POINT2[] " ",TQ_STATE FALSE}
DECL LDAT LL_OLP70={VEL 1.0,ACC 100.0,APO_DIST 50.0,APO_FAC 0.0,ORI_TYP #VAR,CIRC_TYP #BASE,JERK_FAC 50.0}
DECL E6POS Xl021={X 247.672897,Y 971.730774,Z -5.53645706,A -178.005096,B 59.3805809,C -97.2920685,S 2,T 41,E1 0.0,E2 0.0,E3 0.0,E4 0.0,E5 0.0,E6 0.0}
DECL FDAT Fl021={TOOL_NO 2,BASE_NO 3,IPO_FRAME #BASE,POINT2[] " ",TQ_STATE FALSE}
DECL LDAT LL_OLP71={VEL 1.0,ACC 100.0,APO_DIST 50.0,APO_FAC 0.0,ORI_TYP #VAR,CIRC_TYP #BASE,JERK_FAC 50.0}
DECL E6POS Xl026={X 233.621597,Y 967.395508,Z -22.1104393,A -168.154404,B 59.6471596,C -98.7977829,S 2,T 41,E1 0.0,E2 0.0,E3 0.0,E4 0.0,E5 0.0,E6 0.0}
DECL FDAT Fl026={TOOL_NO 2,BASE_NO 3,IPO_FRAME #BASE,POINT2[] " "}
DECL LDAT LL_OLP72={VEL 2.0,ACC 100.0,APO_DIST 0.0,APO_FAC 0.0,ORI_TYP #VAR,CIRC_TYP #BASE,JERK_FAC 50.0}
DECL E6POS XSWP_60_7094={X 221.0009,Y 949.254211,Z -5.67251396,A -158.217896,B 60.0425797,C -90.2032166,S 2,T 41,E1 0.0,E2 0.0,E3 0.0,E4 0.0,E5 0.0,E6 0.0}
DECL FDAT FSWP_60_7094={TOOL_NO 2,BASE_NO 3,IPO_FRAME #BASE,POINT2[] " ",TQ_STATE FALSE}
DECL LDAT LL_OLP73={VEL 2.0,ACC 100.0,APO_DIST 0.0,APO_FAC 0.0,ORI_TYP #VAR,CIRC_TYP #BASE,JERK_FAC 50.0}
DECL E6POS XSWP_60_7092={X 228.085007,Y 955.866516,Z -30.4384708,A -158.172897,B 60.0435295,C -90.218132,S 2,T 41,E1 0.0,E2 0.0,E3 0.0,E4 0.0,E5 0.0,E6 0.0}
DECL FDAT FSWP_60_7092={TOOL_NO 2,BASE_NO 3,IPO_FRAME #BASE,POINT2[] " ",TQ_STATE FALSE}
DECL LDAT LL_OLP74={VEL 2.0,ACC 100.0,APO_DIST 0.0,APO_FAC 0.0,ORI_TYP #VAR,CIRC_TYP #BASE,JERK_FAC 50.0}
DECL E6POS XSWP_60_7090={X 257.39801,Y 968.361877,Z -36.2215195,A -159.207306,B 74.1114807,C -91.3095169,S 2,T 9,E1 0.0,E2 0.0,E3 0.0,E4 0.0,E5 0.0,E6 0.0}
DECL FDAT FSWP_60_7090={TOOL_NO 2,BASE_NO 3,IPO_FRAME #BASE,POINT2[] " ",TQ_STATE FALSE}
DECL LDAT LL_OLP75={VEL 1.0,ACC 100.0,APO_DIST 50.0,APO_FAC 0.0,ORI_TYP #VAR,CIRC_TYP #BASE,JERK_FAC 50.0}
DECL E6POS Xl031={X 272.755188,Y 979.568115,Z -35.2234383,A -159.434296,B 79.5372467,C -93.4828186,S 2,T 9,E1 0.0,E2 0.0,E3 0.0,E4 0.0,E5 0.0,E6 0.0}
DECL FDAT Fl031={TOOL_NO 2,BASE_NO 3,IPO_FRAME #BASE,POINT2[] " ",TQ_STATE FALSE}
DECL LDAT LL_OLP76={VEL 2.0,ACC 100.0,APO_DIST 0.0,APO_FAC 0.0,ORI_TYP #VAR,CIRC_TYP #BASE,JERK_FAC 50.0}
DECL E6POS XSWP_60_7088={X 285.440308,Y 980.615906,Z -43.8656693,A -157.531998,B 82.9950027,C -93.2140198,S 2,T 9,E1 0.0,E2 0.0,E3 0.0,E4 0.0,E5 0.0,E6 0.0}
DECL FDAT FSWP_60_7088={TOOL_NO 2,BASE_NO 3,IPO_FRAME #BASE,POINT2[] " ",TQ_STATE FALSE}
DECL LDAT LL_OLP77={VEL 1.0,ACC 100.0,APO_DIST 50.0,APO_FAC 0.0,ORI_TYP #VAR,CIRC_TYP #BASE,JERK_FAC 50.0}
DECL E6POS Xl036={X 275.141998,Y 983.413818,Z -33.1203995,A 114.270798,B 82.9114609,C 178.523804,S 2,T 9,E1 0.0,E2 0.0,E3 0.0,E4 0.0,E5 0.0,E6 0.0}
DECL FDAT Fl036={TOOL_NO 2,BASE_NO 3,IPO_FRAME #BASE,POINT2[] " ",TQ_STATE FALSE}
DECL LDAT LL_OLP78={VEL 1.0,ACC 100.0,APO_DIST 0.0,APO_FAC 0.0,ORI_TYP #VAR,CIRC_TYP #BASE,JERK_FAC 50.0}
DECL E6POS Xl041={X 252.249496,Y 973.365784,Z -13.6638203,A -178.005096,B 59.3806686,C -97.2922668,S 2,T 41,E1 0.0,E2 0.0,E3 0.0,E4 0.0,E5 0.0,E6 0.0}
DECL FDAT Fl041={TOOL_NO 2,BASE_NO 3,IPO_FRAME #BASE,POINT2[] " "}
DECL LDAT LL_OLP79={VEL 1.0,ACC 100.0,APO_DIST 50.0,APO_FAC 0.0,ORI_TYP #VAR,CIRC_TYP #BASE,JERK_FAC 50.0}
DECL E6POS Xl046={X 295.162598,Y 908.491699,Z -0.105315603,A -179.480606,B 64.3333435,C -98.5977707,S 2,T 41,E1 0.0,E2 0.0,E3 0.0,E4 0.0,E5 0.0,E6 0.0}
DECL FDAT Fl046={TOOL_NO 2,BASE_NO 3,IPO_FRAME #BASE,POINT2[] " "}
DECL PDAT PP_OLP49={VEL 100.0,ACC 100.0,APO_DIST 50.0,APO_MODE #CDIS}
DECL E6POS Xl007={X 640.695679,Y -18.6962795,Z 885.305176,A -143.177597,B 82.1491623,C -143.1194,S 2,T 3,E1 0.0,E2 0.0,E3 0.0,E4 0.0,E5 0.0,E6 0.0}
DECL FDAT Fl007={TOOL_NO 2,BASE_NO 3,IPO_FRAME #BASE,POINT2[] " ",TQ_STATE FALSE}
DECL LDAT LL_OLP82={VEL 2.0,ACC 100.0,APO_DIST 0.0,APO_FAC 0.0,ORI_TYP #VAR,CIRC_TYP #BASE,JERK_FAC 50.0}
DECL E6POS XSWP_60_9560={X 1456.59705,Y 1001.547,Z 327.245514,A -3.69719601,B 74.9993362,C 89.9265213,S 2,T 9,E1 0.0,E2 0.0,E3 0.0,E4 0.0,E5 0.0,E6 0.0}
DECL FDAT FSWP_60_9560={TOOL_NO 2,BASE_NO 3,IPO_FRAME #BASE,POINT2[] " ",TQ_STATE FALSE}
DECL LDAT LL_OLP83={VEL 2.0,ACC 100.0,APO_DIST 0.0,APO_FAC 0.0,ORI_TYP #VAR,CIRC_TYP #BASE,JERK_FAC 50.0}
DECL E6POS XSWP_60_9564={X 1516.00195,Y 996.921692,Z 312.947388,A -3.67799711,B 67.0000992,C 89.9478989,S 2,T 9,E1 0.0,E2 0.0,E3 0.0,E4 0.0,E5 0.0,E6 0.0}
DECL FDAT FSWP_60_9564={TOOL_NO 2,BASE_NO 3,IPO_FRAME #BASE,POINT2[] " ",TQ_STATE FALSE}
DECL LDAT LL_OLP84={VEL 2.0,ACC 100.0,APO_DIST 0.0,APO_FAC 0.0,ORI_TYP #VAR,CIRC_TYP #BASE,JERK_FAC 50.0}
DECL E6POS XSWP_60_9566={X 1547.06201,Y 995.913025,Z 306.494202,A -3.65107489,B 60.0028915,C 89.9666367,S 2,T 9,E1 0.0,E2 0.0,E3 0.0,E4 0.0,E5 0.0,E6 0.0}
DECL FDAT FSWP_60_9566={TOOL_NO 2,BASE_NO 3,IPO_FRAME #BASE,POINT2[] " ",TQ_STATE FALSE}
DECL LDAT LL_OLP88={VEL 2.0,ACC 100.0,APO_DIST 0.0,APO_FAC 0.0,ORI_TYP #VAR,CIRC_TYP #BASE,JERK_FAC 50.0}
DECL E6POS XSWP_60_9565={X 1536.15601,Y -997.677979,Z 299.466614,A 3.67000699,B 60.0004196,C -89.9521408,S 6,T 24,E1 0.0,E2 0.0,E3 0.0,E4 0.0,E5 0.0,E6 0.0}
DECL FDAT FSWP_60_9565={TOOL_NO 2,BASE_NO 3,IPO_FRAME #BASE,POINT2[] " ",TQ_STATE FALSE}
DECL LDAT LL_OLP89={VEL 2.0,ACC 100.0,APO_DIST 0.0,APO_FAC 0.0,ORI_TYP #VAR,CIRC_TYP #BASE,JERK_FAC 50.0}
DECL E6POS XSWP_60_9563={X 1503.87402,Y -998.338684,Z 307.092712,A 3.67000604,B 60.0004196,C -89.9521408,S 6,T 24,E1 0.0,E2 0.0,E3 0.0,E4 0.0,E5 0.0,E6 0.0}
DECL FDAT FSWP_60_9563={TOOL_NO 2,BASE_NO 3,IPO_FRAME #BASE,POINT2[] " ",TQ_STATE FALSE}
DECL LDAT LL_OLP90={VEL 2.0,ACC 100.0,APO_DIST 0.0,APO_FAC 0.0,ORI_TYP #VAR,CIRC_TYP #BASE,JERK_FAC 50.0}
DECL E6POS XSWP_60_9559={X 1451.45398,Y -1007.552,Z 323.418396,A 3.28405404,B 78.6653366,C -90.3185272,S 6,T 24,E1 0.0,E2 0.0,E3 0.0,E4 0.0,E5 0.0,E6 0.0}
DECL FDAT FSWP_60_9559={TOOL_NO 2,BASE_NO 3,IPO_FRAME #BASE,POINT2[] " ",TQ_STATE FALSE}
DECL PDAT PP_OLP56={VEL 100.0,ACC 100.0,APO_DIST 50.0,APO_MODE #CDIS}
DECL E6POS Xl076={X 764.261414,Y -310.796112,Z 1324.02295,A -118.439201,B 84.7641373,C -144.651398,S 2,T 3,E1 0.0,E2 0.0,E3 0.0,E4 0.0,E5 0.0,E6 0.0}
DECL FDAT Fl076={TOOL_NO 2,BASE_NO 3,IPO_FRAME #BASE,POINT2[] " ",TQ_STATE FALSE}
DECL PDAT PP_OLP57={VEL 100.0,ACC 100.0,APO_DIST 50.0,APO_MODE #CDIS}
DECL E6POS Xl008={X 293.173004,Y -908.471985,Z -4.25699997,A 179.468597,B 64.332901,C 98.5838013,S 6,T 24}
DECL FDAT Fl008={TOOL_NO 2,BASE_NO 3,IPO_FRAME #BASE,POINT2[] " ",TQ_STATE FALSE}
DECL LDAT LL_OLP93={VEL 1.0,ACC 100.0,APO_DIST 0.0,APO_FAC 0.0,ORI_TYP #VAR,CIRC_TYP #BASE,JERK_FAC 50.0}
DECL E6POS Xl013={X 247.807602,Y -972.302612,Z -17.5460892,A 178.005005,B 59.3805008,C 97.292099,S 6,T 24,E1 0.0,E2 0.0,E3 0.0,E4 0.0,E5 0.0,E6 0.0}
DECL FDAT Fl013={TOOL_NO 2,BASE_NO 3,IPO_FRAME #BASE,POINT2[] " ",TQ_STATE FALSE}
DECL LDAT LL_OLP94={VEL 1.0,ACC 100.0,APO_DIST 50.0,APO_FAC 0.0,ORI_TYP #VAR,CIRC_TYP #BASE,JERK_FAC 50.0}
DECL E6POS Xl018={X 274.550201,Y -985.772217,Z -39.9958115,A -155.126099,B 79.2151031,C 141.1362,S 6,T 24,E1 0.0,E2 0.0,E3 0.0,E4 0.0,E5 0.0,E6 0.0}
DECL FDAT Fl018={TOOL_NO 2,BASE_NO 3,IPO_FRAME #BASE,POINT2[] " "}
DECL LDAT LL_OLP95={VEL 2.0,ACC 100.0,APO_DIST 0.0,APO_FAC 0.0,ORI_TYP #VAR,CIRC_TYP #BASE,JERK_FAC 50.0}
DECL E6POS XSWP_60_7087={X 282.6185,Y -978.388,Z -47.877121,A 137.080002,B 82.4563904,C 73.1913223,S 2,T 0,E1 0.0,E2 0.0,E3 0.0,E4 0.0,E5 0.0,E6 0.0}
DECL FDAT FSWP_60_7087={TOOL_NO 2,BASE_NO 3,IPO_FRAME #BASE,POINT2[] " ",TQ_STATE FALSE}
DECL LDAT LL_OLP96={VEL 2.0,ACC 100.0,APO_DIST 0.0,APO_FAC 0.0,ORI_TYP #VAR,CIRC_TYP #BASE,JERK_FAC 50.0}
DECL E6POS XSWP_60_7089={X 257.140686,Y -965.624207,Z -42.9535217,A 147.275894,B 69.8397369,C 80.1006165,S 2,T 0,E1 0.0,E2 0.0,E3 0.0,E4 0.0,E5 0.0,E6 0.0}
DECL FDAT FSWP_60_7089={TOOL_NO 2,BASE_NO 3,IPO_FRAME #BASE,POINT2[] " ",TQ_STATE FALSE}
DECL LDAT LL_OLP97={VEL 1.0,ACC 100.0,APO_DIST 50.0,APO_FAC 0.0,ORI_TYP #VAR,CIRC_TYP #BASE,JERK_FAC 50.0}
DECL E6POS Xl023={X 239.181107,Y -960.388,Z -35.9169693,A 158.153702,B 60.04562,C 90.2243805,S 6,T 24,E1 0.0,E2 0.0,E3 0.0,E4 0.0,E5 0.0,E6 0.0}
DECL FDAT Fl023={TOOL_NO 2,BASE_NO 3,IPO_FRAME #BASE,POINT2[] " ",TQ_STATE FALSE}
DECL LDAT LL_OLP98={VEL 2.0,ACC 100.0,APO_DIST 0.0,APO_FAC 0.0,ORI_TYP #VAR,CIRC_TYP #BASE,JERK_FAC 50.0}
DECL E6POS XSWP_60_7091={X 227.981293,Y -953.713623,Z -32.7617302,A 156.240295,B 60.034481,C 88.5653534,S 2,T 0,E1 0.0,E2 0.0,E3 0.0,E4 0.0,E5 0.0,E6 0.0}
DECL FDAT FSWP_60_7091={TOOL_NO 2,BASE_NO 3,IPO_FRAME #BASE,POINT2[] " ",TQ_STATE FALSE}
DECL LDAT LL_OLP99={VEL 2.0,ACC 100.0,APO_DIST 0.0,APO_FAC 0.0,ORI_TYP #VAR,CIRC_TYP #BASE,JERK_FAC 50.0}
DECL E6POS XSWP_60_7093={X 221.411499,Y -949.961792,Z -9.63191605,A 159.264603,B 57.0289192,C 89.6700516,S 2,T 0,E1 0.0,E2 0.0,E3 0.0,E4 0.0,E5 0.0,E6 0.0}
DECL FDAT FSWP_60_7093={TOOL_NO 2,BASE_NO 3,IPO_FRAME #BASE,POINT2[] " ",TQ_STATE FALSE}
DECL LDAT LL_OLP100={VEL 1.0,ACC 100.0,APO_DIST 50.0,APO_FAC 0.0,ORI_TYP #VAR,CIRC_TYP #BASE,JERK_FAC 50.0}
DECL E6POS Xl028={X 239.990097,Y -971.64032,Z -27.5624199,A 168.154297,B 59.6470909,C 98.7976913,S 6,T 24,E1 0.0,E2 0.0,E3 0.0,E4 0.0,E5 0.0,E6 0.0}
DECL FDAT Fl028={TOOL_NO 2,BASE_NO 3,IPO_FRAME #BASE,POINT2[] " ",TQ_STATE FALSE}
DECL LDAT LL_OLP101={VEL 1.0,ACC 100.0,APO_DIST 0.0,APO_FAC 0.0,ORI_TYP #VAR,CIRC_TYP #BASE,JERK_FAC 50.0}
DECL E6POS Xl033={X 248.949203,Y -967.533997,Z -14.2721205,A 178.261505,B 60.3724098,C 97.5146408,S 6,T 24,E1 0.0,E2 0.0,E3 0.0,E4 0.0,E5 0.0,E6 0.0}
DECL FDAT Fl033={TOOL_NO 2,BASE_NO 3,IPO_FRAME #BASE,POINT2[] " "}
DECL LDAT LL_OLP102={VEL 1.0,ACC 100.0,APO_DIST 50.0,APO_FAC 0.0,ORI_TYP #VAR,CIRC_TYP #BASE,JERK_FAC 50.0}
DECL E6POS Xl038={X 293.173004,Y -908.471985,Z -4.25699997,A 179.468597,B 64.332901,C 98.5838013,S 6,T 24}
DECL FDAT Fl038={TOOL_NO 2,BASE_NO 3,IPO_FRAME #BASE,POINT2[] " "}
DECL PDAT PP_OLP58={VEL 100.0,ACC 100.0,APO_DIST 0.0}
DECL E6POS Xl043={X 939.161987,Y -515.692017,Z 1008.57202,A -5.65869999,B 80.3282013,C -85.1673965,S 6,T 27}
DECL FDAT Fl043={TOOL_NO 2,BASE_NO 3,IPO_FRAME #BASE,POINT2[] " ",TQ_STATE FALSE}
DECL PDAT PP_OLP59={VEL 100.0,ACC 100.0,APO_DIST 20.0,APO_MODE #CDIS}
DECL E6POS Xl048={X 1323.32104,Y -409.98999,Z 2256.96509,A 60.4908981,B 73.8983002,C -17.0750999,S 6,T 26}
DECL FDAT Fl048={TOOL_NO 2,BASE_NO 3,IPO_FRAME #BASE,POINT2[] " ",TQ_STATE FALSE}
DECL E6POS XP26={X 1430.43298,Y 920.909485,Z 371.976013,A 50.1822395,B 73.343399,C 129.965698,S 2,T 8,E1 0.0,E2 0.0,E3 0.0,E4 0.0,E5 0.0,E6 0.0}
DECL FDAT FP26={TOOL_NO 2,BASE_NO 3,IPO_FRAME #BASE,POINT2[] " ",TQ_STATE FALSE}
DECL PDAT PPDAT4={VEL 100.0,ACC 100.0,APO_DIST 20.0,APO_MODE #CDIS}
DECL SPOT_SUGG_T LAST_SPOT={GUN[] "1                       ",RETR_CMD[] "#OPN                    ",CHOISE[] "#FIRST                  ",CLO_TM[] "0                       ",PGNO1[] "1                       ",PRESS1[] "0                       ",PGNO2[] "1                       ",PRESS2[] "0                       ",SPOT_PARAMS[] "NORMAL                  "}
DECL E6POS XP27={X 788.400513,Y 515.900818,Z 807.937988,A -165.150604,B 79.6067123,C -105.500099,S 2,T 8,E1 0.0,E2 0.0,E3 0.0,E4 0.0,E5 0.0,E6 0.0}
DECL FDAT FP27={TOOL_NO 2,BASE_NO 3,IPO_FRAME #BASE,POINT2[] " ",TQ_STATE FALSE}
DECL PDAT PPDAT5={VEL 100.0,ACC 100.0,APO_DIST 1.0,APO_MODE #CDIS}
DECL E6POS XP28={X 665.744019,Y -838.904114,Z 179.307205,A -157.579803,B 74.964119,C 117.452499,S 6,T 24,E1 0.0,E2 0.0,E3 0.0,E4 0.0,E5 0.0,E6 0.0}
DECL FDAT FP28={TOOL_NO 2,BASE_NO 3,IPO_FRAME #BASE,POINT2[] " ",TQ_STATE FALSE}
DECL PDAT PPDAT6={VEL 100.0,ACC 100.0,APO_DIST 50.0,APO_MODE #CDIS}
DECL PDAT PP_OLP69={VEL 100.0,ACC 100.0,APO_DIST 100.0,APO_MODE #CDIS}
DECL E6POS Xl062={X 1030.72498,Y 513.461426,Z 1615.24097,A 120.317902,B 17.9576092,C -10.9830999,S 2,T 10,E1 0.0,E2 0.0,E3 0.0,E4 0.0,E5 0.0,E6 0.0}
DECL FDAT Fl062={TOOL_NO 2,BASE_NO 3,IPO_FRAME #BASE,POINT2[] " "}
DECL PDAT PP_OLP70={VEL 100.0,ACC 100.0,APO_DIST 20.0,APO_MODE #CDIS}
DECL E6POS Xl064={X 1807.78406,Y 389.459808,Z 3419.56592,A 63.8189392,B 37.8044701,C -38.9492989,S 2,T 2,E1 0.0,E2 0.0,E3 0.0,E4 0.0,E5 0.0,E6 0.0}
DECL FDAT Fl064={TOOL_NO 2,BASE_NO 3,IPO_FRAME #BASE,POINT2[] " ",TQ_STATE FALSE}
DECL PDAT PP_OLP71={VEL 100.0,ACC 100.0,APO_DIST 20.0,APO_MODE #CDIS}
DECL E6POS Xl067={X 1807.78406,Y 389.459808,Z 3419.56592,A 63.8189392,B 37.8044701,C -38.9492989,S 2,T 2,E1 0.0,E2 0.0,E3 0.0,E4 0.0,E5 0.0,E6 0.0}
DECL FDAT Fl067={TOOL_NO 2,BASE_NO 3,IPO_FRAME #BASE,POINT2[] " ",TQ_STATE FALSE}
DECL E6POS XP29={X 2558.93188,Y -485.116211,Z 3441.69092,A -36.1692314,B -13.5166597,C 1.14306998,S 6,T 27,E1 0.0,E2 0.0,E3 0.0,E4 0.0,E5 0.0,E6 0.0}
DECL FDAT FP29={TOOL_NO 2,BASE_NO 3,IPO_FRAME #BASE,POINT2[] " ",TQ_STATE FALSE}
DECL PDAT PPDAT7={VEL 100.0,ACC 100.0,APO_DIST 50.0,APO_MODE #CDIS}
DECL E6POS XP30={X 2641.70508,Y 753.610291,Z 4294.20215,A 42.6114388,B -30.1368103,C -35.3248711,S 2,T 11,E1 0.0,E2 0.0,E3 0.0,E4 0.0,E5 0.0,E6 0.0}
DECL FDAT FP30={TOOL_NO 2,BASE_NO 3,IPO_FRAME #BASE,POINT2[] " ",TQ_STATE FALSE}
DECL PDAT PPDAT8={VEL 100.0,ACC 100.0,APO_DIST 50.0,APO_MODE #CDIS}
DECL E6POS XP31={X 1807.78699,Y 389.460297,Z 3419.56201,A 63.818779,B 37.8043785,C -38.9489098,S 2,T 2,E1 0.0,E2 0.0,E3 0.0,E4 0.0,E5 0.0,E6 0.0}
DECL FDAT FP31={TOOL_NO 2,BASE_NO 3,IPO_FRAME #BASE,POINT2[] " ",TQ_STATE FALSE}
DECL PDAT PPDAT9={VEL 100.0,ACC 100.0,APO_DIST 50.0,APO_MODE #CDIS}
DECL E6POS XP32={X 978.446411,Y 331.802185,Z 1608.33105,A 19.3579292,B 86.9110107,C 47.965641,S 2,T 10,E1 0.0,E2 0.0,E3 0.0,E4 0.0,E5 0.0,E6 0.0}
DECL FDAT FP32={TOOL_NO 2,BASE_NO 3,IPO_FRAME #BASE,POINT2[] " ",TQ_STATE FALSE}
DECL PDAT PPDAT10={VEL 100.0,ACC 100.0,APO_DIST 50.0,APO_MODE #CDIS}
DECL LDAT LCPDAT22={VEL 2.0,ACC 100.0,APO_DIST 5.0,APO_FAC 50.0,AXIS_VEL 100.0,AXIS_ACC 100.0,ORI_TYP #VAR,CIRC_TYP #BASE,JERK_FAC 50.0,GEAR_JERK 50.0,EXAX_IGN 0}
DECL E6POS XP33={X 1052.75195,Y 58.7190018,Z 2073.41504,A -29.1716995,B 74.7963028,C -24.9258003,S 2,T 3,E1 0.0,E2 0.0,E3 0.0,E4 0.0,E5 0.0,E6 0.0}
DECL FDAT FP33={TOOL_NO 2,BASE_NO 3,IPO_FRAME #BASE,POINT2[] " ",TQ_STATE FALSE}
DECL PDAT PPDAT11={VEL 100.0,ACC 100.0,APO_DIST 50.0,APO_MODE #CDIS}
DECL PDAT PPDAT12={VEL 100.0,ACC 100.0,APO_DIST 100.0,APO_MODE #CDIS}
DECL PDAT PP_OLP72={VEL 100.0,ACC 100.0,APO_DIST 20.0,APO_MODE #CDIS}
DECL E6POS Xl068={X 1080.01196,Y 817.981018,Z 1560.44604,A 110.2062,B 7.66409779,C 0.278902709,S 2,T 10,E1 0.0,E2 0.0,E3 0.0,E4 0.0,E5 0.0,E6 0.0}
DECL FDAT Fl068={TOOL_NO 2,BASE_NO 3,IPO_FRAME #BASE,POINT2[] " "}
DECL PDAT PP_OLP60={VEL 100.0,ACC 100.0,APO_DIST 50.0,APO_MODE #CDIS}
DECL E6POS Xl009={X 336.855988,Y -857.26178,Z 50.4476891,A 179.955597,B 64.2676773,C 108.6987,S 2,T 0,E1 0.0,E2 0.0,E3 0.0,E4 0.0,E5 0.0,E6 0.0}
DECL FDAT Fl009={TOOL_NO 2,BASE_NO 3,IPO_FRAME #BASE,POINT2[] " ",TQ_STATE FALSE}
DECL LDAT LL_OLP103={VEL 1.0,ACC 100.0,APO_DIST 0.0,APO_FAC 0.0,ORI_TYP #VAR,CIRC_TYP #BASE,JERK_FAC 50.0}
DECL E6POS Xl014={X 247.806702,Y -972.302185,Z -17.5459309,A 178.005005,B 59.3804817,C 97.292099,S 2,T 0,E1 0.0,E2 0.0,E3 0.0,E4 0.0,E5 0.0,E6 0.0}
DECL FDAT Fl014={TOOL_NO 2,BASE_NO 3,IPO_FRAME #BASE,POINT2[] " ",TQ_STATE FALSE}
DECL LDAT LL_OLP104={VEL 1.0,ACC 100.0,APO_DIST 50.0,APO_FAC 0.0,ORI_TYP #VAR,CIRC_TYP #BASE,JERK_FAC 50.0}
DECL E6POS Xl019={X 274.548615,Y -985.772095,Z -39.9956017,A -155.126404,B 79.2150726,C 141.135895,S 2,T 0,E1 0.0,E2 0.0,E3 0.0,E4 0.0,E5 0.0,E6 0.0}
DECL FDAT Fl019={TOOL_NO 2,BASE_NO 3,IPO_FRAME #BASE,POINT2[] " "}
DECL LDAT LL_OLP105={VEL 2.0,ACC 100.0,APO_DIST 0.0,APO_FAC 0.0,ORI_TYP #VAR,CIRC_TYP #BASE,JERK_FAC 50.0}
DECL E6POS XSWP_60_7095={X 282.618713,Y -978.388,Z -47.8771286,A 137.079697,B 82.4564667,C 73.1911011,S 2,T 0,E1 0.0,E2 0.0,E3 0.0,E4 0.0,E5 0.0,E6 0.0}
DECL FDAT FSWP_60_7095={TOOL_NO 2,BASE_NO 3,IPO_FRAME #BASE,POINT2[] " ",TQ_STATE FALSE}
DECL LDAT LL_OLP106={VEL 2.0,ACC 100.0,APO_DIST 0.0,APO_FAC 0.0,ORI_TYP #VAR,CIRC_TYP #BASE,JERK_FAC 50.0}
DECL E6POS XSWP_60_7096={X 255.194504,Y -966.905579,Z -47.1379814,A 142.208405,B 69.4559784,C 75.348381,S 2,T 0,E1 0.0,E2 0.0,E3 0.0,E4 0.0,E5 0.0,E6 0.0}
DECL FDAT FSWP_60_7096={TOOL_NO 2,BASE_NO 3,IPO_FRAME #BASE,POINT2[] " ",TQ_STATE FALSE}
DECL LDAT LL_OLP107={VEL 1.0,ACC 100.0,APO_DIST 50.0,APO_FAC 0.0,ORI_TYP #VAR,CIRC_TYP #BASE,JERK_FAC 50.0}
DECL E6POS Xl024={X 239.179398,Y -960.393127,Z -35.9121208,A 158.153702,B 60.045311,C 90.2243118,S 2,T 0,E1 0.0,E2 0.0,E3 0.0,E4 0.0,E5 0.0,E6 0.0}
DECL FDAT Fl024={TOOL_NO 2,BASE_NO 3,IPO_FRAME #BASE,POINT2[] " ",TQ_STATE FALSE}
DECL LDAT LL_OLP108={VEL 2.0,ACC 100.0,APO_DIST 0.0,APO_FAC 0.0,ORI_TYP #VAR,CIRC_TYP #BASE,JERK_FAC 50.0}
DECL E6POS XSWP_60_7097={X 226.203903,Y -955.712891,Z -37.8997803,A 152.657898,B 59.94104,C 85.4634781,S 2,T 0,E1 0.0,E2 0.0,E3 0.0,E4 0.0,E5 0.0,E6 0.0}
DECL FDAT FSWP_60_7097={TOOL_NO 2,BASE_NO 3,IPO_FRAME #BASE,POINT2[] " ",TQ_STATE FALSE}
DECL LDAT LL_OLP109={VEL 2.0,ACC 100.0,APO_DIST 0.0,APO_FAC 0.0,ORI_TYP #VAR,CIRC_TYP #BASE,JERK_FAC 50.0}
DECL E6POS XSWP_60_7098={X 220.989105,Y -950.801514,Z -16.8052597,A 158.216995,B 59.2779617,C 88.5233002,S 2,T 0,E1 0.0,E2 0.0,E3 0.0,E4 0.0,E5 0.0,E6 0.0}
DECL FDAT FSWP_60_7098={TOOL_NO 2,BASE_NO 3,IPO_FRAME #BASE,POINT2[] " ",TQ_STATE FALSE}
DECL LDAT LL_OLP110={VEL 1.0,ACC 100.0,APO_DIST 50.0,APO_FAC 0.0,ORI_TYP #VAR,CIRC_TYP #BASE,JERK_FAC 50.0}
DECL E6POS Xl029={X 239.989304,Y -971.639771,Z -27.5622807,A 168.154297,B 59.6470795,C 98.797699,S 2,T 0,E1 0.0,E2 0.0,E3 0.0,E4 0.0,E5 0.0,E6 0.0}
DECL FDAT Fl029={TOOL_NO 2,BASE_NO 3,IPO_FRAME #BASE,POINT2[] " ",TQ_STATE FALSE}
DECL LDAT LL_OLP111={VEL 1.0,ACC 100.0,APO_DIST 0.0,APO_FAC 0.0,ORI_TYP #VAR,CIRC_TYP #BASE,JERK_FAC 50.0}
DECL E6POS Xl034={X 248.944397,Y -967.534302,Z -14.2736702,A 178.261398,B 60.3724709,C 97.514679,S 2,T 0,E1 0.0,E2 0.0,E3 0.0,E4 0.0,E5 0.0,E6 0.0}
DECL FDAT Fl034={TOOL_NO 2,BASE_NO 3,IPO_FRAME #BASE,POINT2[] " "}
DECL LDAT LL_OLP112={VEL 1.0,ACC 100.0,APO_DIST 50.0,APO_FAC 0.0,ORI_TYP #VAR,CIRC_TYP #BASE,JERK_FAC 50.0}
DECL E6POS Xl039={X 293.158813,Y -908.473083,Z -4.27368307,A 179.468201,B 64.3345795,C 98.5854263,S 2,T 0,E1 0.0,E2 0.0,E3 0.0,E4 0.0,E5 0.0,E6 0.0}
DECL FDAT Fl039={TOOL_NO 2,BASE_NO 3,IPO_FRAME #BASE,POINT2[] " "}
DECL PDAT PP_OLP61={VEL 100.0,ACC 100.0,APO_DIST 0.0}
DECL E6POS Xl044={X 938.180481,Y -515.384827,Z 748.889771,A 158.332504,B 85.8407593,C 83.1708679,S 2,T 1,E1 0.0,E2 0.0,E3 0.0,E4 0.0,E5 0.0,E6 0.0}
DECL FDAT Fl044={TOOL_NO 2,BASE_NO 3,IPO_FRAME #BASE,POINT2[] " ",TQ_STATE FALSE}
DECL PDAT PP_OLP62={VEL 100.0,ACC 100.0,APO_DIST 20.0,APO_MODE #CDIS}
DECL E6POS Xl049={X 640.695679,Y -18.6962795,Z 885.305176,A -143.177597,B 82.1491623,C -143.1194,S 2,T 3,E1 0.0,E2 0.0,E3 0.0,E4 0.0,E5 0.0,E6 0.0}
DECL FDAT Fl049={TOOL_NO 2,BASE_NO 3,IPO_FRAME #BASE,POINT2[] " ",TQ_STATE FALSE}
DECL E6POS XP1={X 764.261414,Y -310.796112,Z 1324.02295,A -118.439201,B 84.7641373,C -144.651398,S 2,T 3,E1 0.0,E2 0.0,E3 0.0,E4 0.0,E5 0.0,E6 0.0}
DECL FDAT FP1={TOOL_NO 2,BASE_NO 3,IPO_FRAME #BASE,POINT2[] " ",TQ_STATE FALSE}
DECL PDAT PPDAT1={VEL 100.0,ACC 100.0,APO_DIST 50.0,APO_MODE #CDIS}
DECL LDAT LCPDAT1={VEL 2.0,ACC 100.0,APO_DIST 100.0,APO_FAC 50.0,AXIS_VEL 100.0,AXIS_ACC 100.0,ORI_TYP #VAR,CIRC_TYP #BASE,JERK_FAC 50.0,GEAR_JERK 50.0,EXAX_IGN 0}
DECL PDAT PPDAT2={VEL 100.0,ACC 100.0,APO_DIST 50.0,APO_MODE #CDIS}
DECL LDAT LCPDAT2={VEL 2.0,ACC 100.0,APO_DIST 100.0,APO_FAC 50.0,AXIS_VEL 100.0,AXIS_ACC 100.0,ORI_TYP #VAR,CIRC_TYP #BASE,JERK_FAC 50.0,GEAR_JERK 50.0,EXAX_IGN 0}
DECL PDAT PPDAT3={VEL 100.0,ACC 100.0,APO_DIST 50.0,APO_MODE #CDIS}
DECL LDAT LCPDAT3={VEL 2.0,ACC 100.0,APO_DIST 100.0,APO_FAC 50.0,AXIS_VEL 100.0,AXIS_ACC 100.0,ORI_TYP #VAR,CIRC_TYP #BASE,JERK_FAC 50.0,GEAR_JERK 50.0,EXAX_IGN 0}
DECL PDAT PPDAT13={VEL 100.0,ACC 100.0,APO_DIST 50.0,APO_MODE #CDIS}
DECL LDAT LCPDAT4={VEL 2.0,ACC 100.0,APO_DIST 100.0,APO_FAC 50.0,AXIS_VEL 100.0,AXIS_ACC 100.0,ORI_TYP #VAR,CIRC_TYP #BASE,JERK_FAC 50.0,GEAR_JERK 50.0,EXAX_IGN 0}
DECL PDAT PPDAT14={VEL 100.0,ACC 100.0,APO_DIST 50.0,APO_MODE #CDIS}
DECL PDAT PPDAT15={VEL 100.0,ACC 100.0,APO_DIST 20.0,APO_MODE #CDIS}
DECL LDAT LCPDAT5={VEL 2.0,ACC 100.0,APO_DIST 0.0,APO_FAC 50.0,AXIS_VEL 100.0,AXIS_ACC 100.0,ORI_TYP #VAR,CIRC_TYP #BASE,JERK_FAC 50.0,GEAR_JERK 50.0,EXAX_IGN 0}
DECL PDAT PPDAT16={VEL 100.0,ACC 100.0,APO_DIST 20.0,APO_MODE #CDIS}
DECL LDAT LCPDAT6={VEL 2.0,ACC 100.0,APO_DIST 50.0,APO_FAC 50.0,AXIS_VEL 100.0,AXIS_ACC 100.0,ORI_TYP #VAR,CIRC_TYP #BASE,JERK_FAC 50.0,GEAR_JERK 50.0,EXAX_IGN 0}
DECL PDAT PPDAT17={VEL 100.0,ACC 100.0,APO_DIST 50.0,APO_MODE #CDIS}
DECL LDAT LCPDAT7={VEL 2.0,ACC 100.0,APO_DIST 100.0,APO_FAC 50.0,AXIS_VEL 100.0,AXIS_ACC 100.0,ORI_TYP #VAR,CIRC_TYP #BASE,JERK_FAC 50.0,GEAR_JERK 50.0,EXAX_IGN 0}
DECL PDAT PPDAT18={VEL 100.0,ACC 100.0,APO_DIST 50.0,APO_MODE #CDIS}
DECL LDAT LCPDAT8={VEL 2.0,ACC 100.0,APO_DIST 100.0,APO_FAC 50.0,AXIS_VEL 100.0,AXIS_ACC 100.0,ORI_TYP #VAR,CIRC_TYP #BASE,JERK_FAC 50.0,GEAR_JERK 50.0,EXAX_IGN 0}
DECL PDAT PPDAT19={VEL 100.0,ACC 100.0,APO_DIST 20.0,APO_MODE #CDIS}
DECL LDAT LCPDAT9={VEL 2.0,ACC 100.0,APO_DIST 50.0,APO_FAC 50.0,AXIS_VEL 100.0,AXIS_ACC 100.0,ORI_TYP #VAR,CIRC_TYP #BASE,JERK_FAC 50.0,GEAR_JERK 50.0,EXAX_IGN 0}
DECL PDAT PPDAT20={VEL 100.0,ACC 100.0,APO_DIST 50.0,APO_MODE #CDIS}
DECL LDAT LCPDAT10={VEL 2.0,ACC 100.0,APO_DIST 100.0,APO_FAC 50.0,AXIS_VEL 100.0,AXIS_ACC 100.0,ORI_TYP #VAR,CIRC_TYP #BASE,JERK_FAC 50.0,GEAR_JERK 50.0,EXAX_IGN 0}
DECL PDAT PPDAT21={VEL 100.0,ACC 100.0,APO_DIST 50.0,APO_MODE #CDIS}
DECL LDAT LCPDAT11={VEL 2.0,ACC 100.0,APO_DIST 100.0,APO_FAC 50.0,AXIS_VEL 100.0,AXIS_ACC 100.0,ORI_TYP #VAR,CIRC_TYP #BASE,JERK_FAC 50.0,GEAR_JERK 50.0,EXAX_IGN 0}
DECL PDAT PPDAT22={VEL 100.0,ACC 100.0,APO_DIST 20.0,APO_MODE #CDIS}
DECL LDAT LCPDAT12={VEL 2.0,ACC 100.0,APO_DIST 50.0,APO_FAC 50.0,AXIS_VEL 100.0,AXIS_ACC 100.0,ORI_TYP #VAR,CIRC_TYP #BASE,JERK_FAC 50.0,GEAR_JERK 50.0,EXAX_IGN 0}
DECL PDAT PPDAT23={VEL 100.0,ACC 100.0,APO_DIST 20.0,APO_MODE #CDIS}
DECL LDAT LCPDAT13={VEL 2.0,ACC 100.0,APO_DIST 0.0,APO_FAC 50.0,AXIS_VEL 100.0,AXIS_ACC 100.0,ORI_TYP #VAR,CIRC_TYP #BASE,JERK_FAC 50.0,GEAR_JERK 50.0,EXAX_IGN 0}
DECL PDAT PPDAT24={VEL 100.0,ACC 100.0,APO_DIST 20.0,APO_MODE #CDIS}
DECL LDAT LCPDAT14={VEL 2.0,ACC 100.0,APO_DIST 50.0,APO_FAC 50.0,AXIS_VEL 100.0,AXIS_ACC 100.0,ORI_TYP #VAR,CIRC_TYP #BASE,JERK_FAC 50.0,GEAR_JERK 50.0,EXAX_IGN 0}
DECL PDAT PPDAT25={VEL 100.0,ACC 100.0,APO_DIST 50.0,APO_MODE #CDIS}
DECL LDAT LCPDAT15={VEL 2.0,ACC 100.0,APO_DIST 100.0,APO_FAC 50.0,AXIS_VEL 100.0,AXIS_ACC 100.0,ORI_TYP #VAR,CIRC_TYP #BASE,JERK_FAC 50.0,GEAR_JERK 50.0,EXAX_IGN 0}
DECL PDAT PPDAT26={VEL 100.0,ACC 100.0,APO_DIST 20.0,APO_MODE #CDIS}
DECL LDAT LCPDAT16={VEL 2.0,ACC 100.0,APO_DIST 50.0,APO_FAC 50.0,AXIS_VEL 100.0,AXIS_ACC 100.0,ORI_TYP #VAR,CIRC_TYP #BASE,JERK_FAC 50.0,GEAR_JERK 50.0,EXAX_IGN 0}
DECL PDAT PPDAT27={VEL 100.0,ACC 100.0,APO_DIST 20.0,APO_MODE #CDIS}
DECL LDAT LCPDAT17={VEL 2.0,ACC 100.0,APO_DIST 50.0,APO_FAC 50.0,AXIS_VEL 100.0,AXIS_ACC 100.0,ORI_TYP #VAR,CIRC_TYP #BASE,JERK_FAC 50.0,GEAR_JERK 50.0,EXAX_IGN 0}
DECL PDAT PPDAT28={VEL 100.0,ACC 100.0,APO_DIST 20.0,APO_MODE #CDIS}
DECL LDAT LCPDAT18={VEL 2.0,ACC 100.0,APO_DIST 50.0,APO_FAC 50.0,AXIS_VEL 100.0,AXIS_ACC 100.0,ORI_TYP #VAR,CIRC_TYP #BASE,JERK_FAC 50.0,GEAR_JERK 50.0,EXAX_IGN 0}
DECL PDAT PPDAT29={VEL 100.0,ACC 100.0,APO_DIST 50.0,APO_MODE #CDIS}
DECL LDAT LCPDAT19={VEL 2.0,ACC 100.0,APO_DIST 100.0,APO_FAC 50.0,AXIS_VEL 100.0,AXIS_ACC 100.0,ORI_TYP #VAR,CIRC_TYP #BASE,JERK_FAC 50.0,GEAR_JERK 50.0,EXAX_IGN 0}
DECL PDAT PPDAT30={VEL 100.0,ACC 100.0,APO_DIST 50.0,APO_MODE #CDIS}
DECL LDAT LCPDAT20={VEL 2.0,ACC 100.0,APO_DIST 100.0,APO_FAC 50.0,AXIS_VEL 100.0,AXIS_ACC 100.0,ORI_TYP #VAR,CIRC_TYP #BASE,JERK_FAC 50.0,GEAR_JERK 50.0,EXAX_IGN 0}
DECL PDAT PPDAT31={VEL 100.0,ACC 100.0,APO_DIST 50.0,APO_MODE #CDIS}
DECL LDAT LCPDAT21={VEL 2.0,ACC 100.0,APO_DIST 100.0,APO_FAC 50.0,AXIS_VEL 100.0,AXIS_ACC 100.0,ORI_TYP #VAR,CIRC_TYP #BASE,JERK_FAC 50.0,GEAR_JERK 50.0,EXAX_IGN 0}
DECL PDAT PPDAT32={VEL 100.0,ACC 100.0,APO_DIST 50.0,APO_MODE #CDIS}
DECL LDAT LCPDAT23={VEL 2.0,ACC 100.0,APO_DIST 100.0,APO_FAC 50.0,AXIS_VEL 100.0,AXIS_ACC 100.0,ORI_TYP #VAR,CIRC_TYP #BASE,JERK_FAC 50.0,GEAR_JERK 50.0,EXAX_IGN 0}
DECL PDAT PPDAT33={VEL 100.0,ACC 100.0,APO_DIST 20.0,APO_MODE #CDIS}
DECL LDAT LCPDAT24={VEL 2.0,ACC 100.0,APO_DIST 50.0,APO_FAC 50.0,AXIS_VEL 100.0,AXIS_ACC 100.0,ORI_TYP #VAR,CIRC_TYP #BASE,JERK_FAC 50.0,GEAR_JERK 50.0,EXAX_IGN 0}
DECL PDAT PPDAT34={VEL 100.0,ACC 100.0,APO_DIST 50.0,APO_MODE #CDIS}
DECL LDAT LCPDAT25={VEL 2.0,ACC 100.0,APO_DIST 100.0,APO_FAC 50.0,AXIS_VEL 100.0,AXIS_ACC 100.0,ORI_TYP #VAR,CIRC_TYP #BASE,JERK_FAC 50.0,GEAR_JERK 50.0,EXAX_IGN 0}
DECL PDAT PPDAT35={VEL 100.0,ACC 100.0,APO_DIST 20.0,APO_MODE #CDIS}
DECL LDAT LCPDAT26={VEL 2.0,ACC 100.0,APO_DIST 50.0,APO_FAC 50.0,AXIS_VEL 100.0,AXIS_ACC 100.0,ORI_TYP #VAR,CIRC_TYP #BASE,JERK_FAC 50.0,GEAR_JERK 50.0,EXAX_IGN 0}
DECL PDAT PPDAT36={VEL 100.0,ACC 100.0,APO_DIST 20.0,APO_MODE #CDIS}
DECL LDAT LCPDAT27={VEL 2.0,ACC 100.0,APO_DIST 0.0,APO_FAC 50.0,AXIS_VEL 100.0,AXIS_ACC 100.0,ORI_TYP #VAR,CIRC_TYP #BASE,JERK_FAC 50.0,GEAR_JERK 50.0,EXAX_IGN 0}
DECL PDAT PPDAT37={VEL 100.0,ACC 100.0,APO_DIST 20.0,APO_MODE #CDIS}
DECL LDAT LCPDAT28={VEL 2.0,ACC 100.0,APO_DIST 50.0,APO_FAC 50.0,AXIS_VEL 100.0,AXIS_ACC 100.0,ORI_TYP #VAR,CIRC_TYP #BASE,JERK_FAC 50.0,GEAR_JERK 50.0,EXAX_IGN 0}
DECL PDAT Pxlarge={VEL 100.0,ACC 100.0,APO_DIST 500.0,APO_MODE #CDIS}
DECL E6POS XP0={X 1807.78296,Y 389.460297,Z 3419.56494,A 63.8189697,B 37.8044815,C -38.9492798,S 2,T 2,E1 0.0,E2 0.0,E3 0.0,E4 0.0,E5 0.0,E6 0.0}
DECL FDAT FP0={TOOL_NO 2,BASE_NO 3,IPO_FRAME #BASE,POINT2[] " ",TQ_STATE FALSE}
DECL PDAT Pvmax={VEL 100.0,ACC 100.0,APO_DIST 50.0,APO_MODE #CDIS}
DECL E6POS Xl012={X 1110.92896,Y 490.82251,Z 1769.04504,A 121.191299,B 20.5780697,C -14.8572798,S 2,T 10,E1 0.0,E2 0.0,E3 0.0,E4 0.0,E5 0.0,E6 0.0}
DECL FDAT Fl012={TOOL_NO 2,BASE_NO 3,IPO_FRAME #BASE,POINT2[] " ",TQ_STATE FALSE}
DECL PDAT Pmedium={VEL 100.0,ACC 100.0,APO_DIST 100.0,APO_MODE #CDIS}
DECL E6POS Xl017={X 864.710083,Y 543.601685,Z 1541.43604,A 120.7864,B 15.0748196,C -6.08685398,S 2,T 10,E1 0.0,E2 0.0,E3 0.0,E4 0.0,E5 0.0,E6 0.0}
DECL FDAT Fl017={TOOL_NO 2,BASE_NO 3,IPO_FRAME #BASE,POINT2[] " "}
DECL PDAT Pfin={VEL 100.0,ACC 100.0,APO_DIST 20.0,APO_MODE #CDIS}
DECL E6POS Xl022={X 641.701477,Y 906.07019,Z 1473.96704,A 121.870697,B 10.4103603,C -1.61694098,S 2,T 10,E1 0.0,E2 0.0,E3 0.0,E4 0.0,E5 0.0,E6 0.0}
DECL FDAT Fl022={TOOL_NO 2,BASE_NO 3,IPO_FRAME #BASE,POINT2[] " ",TQ_STATE FALSE}
DECL E6POS Xl027={X 641.701477,Y 906.07019,Z 1473.96704,A 121.870697,B 10.4103603,C -1.61694098,S 2,T 10,E1 0.0,E2 0.0,E3 0.0,E4 0.0,E5 0.0,E6 0.0}
DECL FDAT Fl027={TOOL_NO 2,BASE_NO 3,IPO_FRAME #BASE,POINT2[] " ",TQ_STATE FALSE}
DECL PDAT Psmall={VEL 100.0,ACC 100.0,APO_DIST 50.0,APO_MODE #CDIS}
DECL E6POS Xl065={X 699.777222,Y 845.145081,Z 1471.58203,A 112.012901,B 10.4008102,C -1.17845297,S 2,T 10,E1 0.0,E2 0.0,E3 0.0,E4 0.0,E5 0.0,E6 0.0}
DECL FDAT Fl065={TOOL_NO 2,BASE_NO 3,IPO_FRAME #BASE,POINT2[] " "}
DECL E6POS Xl066={X 888.990417,Y 837.006226,Z 1554.802,A 109.171799,B 9.07432747,C -3.06951308,S 2,T 10,E1 0.0,E2 0.0,E3 0.0,E4 0.0,E5 0.0,E6 0.0}
DECL FDAT Fl066={TOOL_NO 2,BASE_NO 3,IPO_FRAME #BASE,POINT2[] " "}
DECL E6POS Xl081={X 1098.56995,Y 846.792419,Z 1500.58105,A 102.1334,B 7.67785501,C -0.307278514,S 2,T 10,E1 0.0,E2 0.0,E3 0.0,E4 0.0,E5 0.0,E6 0.0}
DECL FDAT Fl081={TOOL_NO 2,BASE_NO 3,IPO_FRAME #BASE,POINT2[] " "}
DECL E6POS Xl096={X 1244.01501,Y 880.145813,Z 1504.479,A 93.5144119,B 7.09015083,C 0.0830439627,S 2,T 10,E1 0.0,E2 0.0,E3 0.0,E4 0.0,E5 0.0,E6 0.0}
DECL FDAT Fl096={TOOL_NO 2,BASE_NO 3,IPO_FRAME #BASE,POINT2[] " "}
DECL E6POS Xl106={X 1244.01294,Y 880.152771,Z 1504.479,A 93.5145874,B 7.09015083,C 0.082997933,S 2,T 10,E1 0.0,E2 0.0,E3 0.0,E4 0.0,E5 0.0,E6 0.0}
DECL FDAT Fl106={TOOL_NO 2,BASE_NO 3,IPO_FRAME #BASE,POINT2[] " ",TQ_STATE FALSE}
DECL PDAT Plarge={VEL 100.0,ACC 100.0,APO_DIST 200.0,APO_MODE #CDIS}
DECL E6POS Xl111={X 1195.76099,Y 769.465271,Z 1465.20203,A 77.7666626,B 8.78154469,C 19.8225403,S 2,T 10,E1 0.0,E2 0.0,E3 0.0,E4 0.0,E5 0.0,E6 0.0}
DECL FDAT Fl111={TOOL_NO 2,BASE_NO 3,IPO_FRAME #BASE,POINT2[] " "}
DECL E6POS Xl116={X 1216.97095,Y 589.121582,Z 1381.71899,A 34.8473587,B 42.6439514,C 68.814827,S 2,T 10,E1 0.0,E2 0.0,E3 0.0,E4 0.0,E5 0.0,E6 0.0}
DECL FDAT Fl116={TOOL_NO 2,BASE_NO 3,IPO_FRAME #BASE,POINT2[] " ",TQ_STATE FALSE}
DECL E6POS Xl126={X 1102.81799,Y 658.877808,Z 901.249817,A 51.5279808,B 70.0681381,C 126.176102,S 2,T 8,E1 0.0,E2 0.0,E3 0.0,E4 0.0,E5 0.0,E6 0.0}
DECL FDAT Fl126={TOOL_NO 2,BASE_NO 3,IPO_FRAME #BASE,POINT2[] " "}
DECL E6POS Xl131={X 1430.453,Y 920.916016,Z 371.963989,A 61.0419998,B 56.5774002,C 153.318497,S 2,T 8}
DECL FDAT Fl131={TOOL_NO 2,BASE_NO 3,IPO_FRAME #BASE,POINT2[] " ",TQ_STATE FALSE}
DECL LDAT LL_OLP12={VEL 1.0,ACC 100.0,APO_DIST 50.0,APO_FAC 0.0,ORI_TYP #VAR,CIRC_TYP #BASE,JERK_FAC 50.0}
DECL E6POS Xl136={X 1430.48706,Y 1010.909,Z 362.902008,A 62.6833992,B 57.0157089,C 154.692001,S 2,T 8,E1 0.0,E2 0.0,E3 0.0,E4 0.0,E5 0.0,E6 0.0}
DECL FDAT Fl136={TOOL_NO 2,BASE_NO 3,IPO_FRAME #BASE,POINT2[] " "}
DECL LDAT LL_OLP13={VEL 1.0,ACC 100.0,APO_DIST 50.0,APO_FAC 0.0,ORI_TYP #VAR,CIRC_TYP #BASE,JERK_FAC 50.0}
DECL E6POS Xl140={X 1436.12805,Y 1016.59003,Z 346.825104,A 60.8482018,B 67.7460022,C 152.708603,S 2,T 8,E1 0.0,E2 0.0,E3 0.0,E4 0.0,E5 0.0,E6 0.0}
DECL FDAT Fl140={TOOL_NO 2,BASE_NO 3,IPO_FRAME #BASE,POINT2[] " "}
DECL LDAT LL_OLP23={VEL 1.0,ACC 100.0,APO_DIST 50.0,APO_FAC 0.0,ORI_TYP #VAR,CIRC_TYP #BASE,JERK_FAC 50.0}
DECL E6POS Xl145={X 1419.27002,Y 1007.05603,Z 328.158997,A 42.0032997,B 86.8728027,C 142.518997,S 2,T 9}
DECL FDAT Fl145={TOOL_NO 2,BASE_NO 3,IPO_FRAME #BASE,POINT2[] " "}
DECL E6POS Xl107={X 1287.51099,Y 815.0401,Z 1505.87903,A 91.2015533,B 7.43633413,C 0.250840098,S 2,T 10,E1 0.0,E2 0.0,E3 0.0,E4 0.0,E5 0.0,E6 0.0}
DECL FDAT Fl107={TOOL_NO 2,BASE_NO 3,IPO_FRAME #BASE,POINT2[] " ",TQ_STATE FALSE}
DECL E6POS Xl117={X 1467.48499,Y 499.312988,Z 1128.79102,A 24.08284,B 48.1840591,C 76.8556671,S 2,T 10,E1 0.0,E2 0.0,E3 0.0,E4 0.0,E5 0.0,E6 0.0}
DECL FDAT Fl117={TOOL_NO 2,BASE_NO 3,IPO_FRAME #BASE,POINT2[] " "}
DECL E6POS Xl127={X 1472.69604,Y 897.264282,Z 388.649597,A 52.5739784,B 66.1850433,C 142.9823,S 2,T 8,E1 0.0,E2 0.0,E3 0.0,E4 0.0,E5 0.0,E6 0.0}
DECL FDAT Fl127={TOOL_NO 2,BASE_NO 3,IPO_FRAME #BASE,POINT2[] " "}
DECL E6POS Xl132={X 1434.48706,Y 1005.49799,Z 362.049988,A 57.4928093,B 67.308403,C 146.797607,S 2,T 8,E1 0.0,E2 0.0,E3 0.0,E4 0.0,E5 0.0,E6 0.0}
DECL FDAT Fl132={TOOL_NO 2,BASE_NO 3,IPO_FRAME #BASE,POINT2[] " ",TQ_STATE FALSE}
DECL E6POS Xl133={X 1442.87402,Y 1010.96802,Z 348.503601,A 104.2127,B 77.6701736,C -159.955597,S 2,T 9,E1 0.0,E2 0.0,E3 0.0,E4 0.0,E5 0.0,E6 0.0}
DECL FDAT Fl133={TOOL_NO 2,BASE_NO 3,IPO_FRAME #BASE,POINT2[] " ",TQ_STATE FALSE}
DECL LDAT LL_OLP56={VEL 1.0,ACC 100.0,APO_DIST 5.0,APO_FAC 0.0,ORI_TYP #VAR,CIRC_TYP #BASE,JERK_FAC 50.0}
DECL E6POS Xl151={X 1482.73804,Y 1005.48102,Z 342.670685,A 40.8555908,B 61.7790604,C 132.761597,S 2,T 8,E1 0.0,E2 0.0,E3 0.0,E4 0.0,E5 0.0,E6 0.0}
DECL FDAT Fl151={TOOL_NO 2,BASE_NO 3,IPO_FRAME #BASE,POINT2[] " ",TQ_STATE FALSE}
DECL E6POS Xl156={X 1471.53406,Y 995.791016,Z 370.27301,A 40.8555908,B 61.7790604,C 132.761597,S 2,T 8,E1 0.0,E2 0.0,E3 0.0,E4 0.0,E5 0.0,E6 0.0}
DECL FDAT Fl156={TOOL_NO 2,BASE_NO 3,IPO_FRAME #BASE,POINT2[] " "}
DECL PDAT PPDAT0={VEL 100.0,ACC 100.0,APO_DIST 20.0,APO_MODE #CDIS}
DECL E6POS XP2={X 1632.59497,Y 898.653381,Z 347.892609,A 29.9060497,B 62.699501,C 131.190002,S 2,T 8,E1 0.0,E2 0.0,E3 0.0,E4 0.0,E5 0.0,E6 0.0}
DECL FDAT FP2={TOOL_NO 2,BASE_NO 3,IPO_FRAME #BASE,POINT2[] " ",TQ_STATE FALSE}
DECL E6POS Xl166={X 2158.54199,Y 932.498413,Z 299.678802,A 90.0003281,B 50.0004311,C -89.9996719,S 2,T 41,E1 0.0,E2 0.0,E3 0.0,E4 0.0,E5 0.0,E6 0.0}
DECL FDAT Fl166={TOOL_NO 2,BASE_NO 3,IPO_FRAME #BASE,POINT2[] " "}
DECL E6POS Xl171={X 2211.60205,Y 932.498718,Z 299.678894,A 90.0003204,B 50.0004311,C -89.9996872,S 2,T 41,E1 0.0,E2 0.0,E3 0.0,E4 0.0,E5 0.0,E6 0.0}
DECL FDAT Fl171={TOOL_NO 2,BASE_NO 3,IPO_FRAME #BASE,POINT2[] " ",TQ_STATE FALSE}
DECL E6POS Xl176={X 2208.22998,Y 950.995178,Z 277.635315,A 91.9777832,B 49.9836311,C -88.4849701,S 2,T 41,E1 0.0,E2 0.0,E3 0.0,E4 0.0,E5 0.0,E6 0.0}
DECL FDAT Fl176={TOOL_NO 2,BASE_NO 3,IPO_FRAME #BASE,POINT2[] " "}
DECL LDAT Lsmall={VEL 2.0,ACC 100.0,APO_DIST 5.0,APO_FAC 50.0,AXIS_VEL 100.0,AXIS_ACC 100.0,ORI_TYP #VAR,CIRC_TYP #BASE,JERK_FAC 50.0,GEAR_JERK 50.0,EXAX_IGN 0}
DECL E6POS Xl181={X 2208.22412,Y 951.037781,Z 277.642487,A 91.9245682,B 49.9830513,C -88.5262527,S 2,T 41,E1 0.0,E2 0.0,E3 0.0,E4 0.0,E5 0.0,E6 0.0}
DECL FDAT Fl181={TOOL_NO 2,BASE_NO 3,IPO_FRAME #BASE,POINT2[] " ",TQ_STATE FALSE}
DECL LDAT LL_OLP63={VEL 1.0,ACC 100.0,APO_DIST 5.0,APO_FAC 0.0,ORI_TYP #VAR,CIRC_TYP #BASE,JERK_FAC 50.0}
DECL E6POS Xl196={X 2205.21704,Y 709.570007,Z 304.463013,A 90.0,B 70.0,C -90.0,S 2,T 41}
DECL FDAT Fl196={TOOL_NO 2,BASE_NO 3,IPO_FRAME #BASE,POINT2[] " "}
DECL LDAT LL_OLP64={VEL 1.0,ACC 100.0,APO_DIST 5.0,APO_FAC 0.0,ORI_TYP #VAR,CIRC_TYP #BASE,JERK_FAC 50.0}
DECL E6POS Xl201={X 2211.9541,Y 610.777588,Z 321.752991,A 115.6633,B 81.5526733,C -64.4972763,S 2,T 9,E1 0.0,E2 0.0,E3 0.0,E4 0.0,E5 0.0,E6 0.0}
DECL FDAT Fl201={TOOL_NO 2,BASE_NO 3,IPO_FRAME #BASE,POINT2[] " "}
DECL LDAT LL_OLP65={VEL 1.0,ACC 100.0,APO_DIST 30.0,APO_FAC 0.0,ORI_TYP #VAR,CIRC_TYP #BASE,JERK_FAC 50.0}
DECL E6POS Xl206={X 2210.24512,Y 588.605408,Z 326.740112,A 135.544601,B 82.8303375,C -44.6895409,S 2,T 9,E1 0.0,E2 0.0,E3 0.0,E4 0.0,E5 0.0,E6 0.0}
DECL FDAT Fl206={TOOL_NO 2,BASE_NO 3,IPO_FRAME #BASE,POINT2[] " ",TQ_STATE FALSE}
DECL LDAT LL_OLP66={VEL 1.0,ACC 100.0,APO_DIST 1.0,APO_FAC 0.0,ORI_TYP #VAR,CIRC_TYP #BASE,JERK_FAC 50.0}
DECL E6POS Xl216={X 2212.45605,Y 338.983887,Z 469.024414,A -152.774597,B 84.9349136,C 27.8669205,S 2,T 9,E1 0.0,E2 0.0,E3 0.0,E4 0.0,E5 0.0,E6 0.0}
DECL FDAT Fl216={TOOL_NO 2,BASE_NO 3,IPO_FRAME #BASE,POINT2[] " "}
DECL PDAT PPDAT38={VEL 100.0,ACC 100.0,APO_DIST 50.0,APO_MODE #CDIS}
DECL E6POS Xl221={X 2212.71411,Y 294.405914,Z 491.214996,A -98.7656631,B 84.3133469,C 81.4460602,S 2,T 9,E1 0.0,E2 0.0,E3 0.0,E4 0.0,E5 0.0,E6 0.0}
DECL FDAT Fl221={TOOL_NO 2,BASE_NO 3,IPO_FRAME #BASE,POINT2[] " ",TQ_STATE FALSE}
DECL PDAT PPDAT39={VEL 100.0,ACC 100.0,APO_DIST 50.0,APO_MODE #CDIS}
DECL E6POS Xl226={X 2214.04907,Y 167.135101,Z 494.44339,A -88.2585373,B 76.3280487,C 91.5829697,S 2,T 9,E1 0.0,E2 0.0,E3 0.0,E4 0.0,E5 0.0,E6 0.0}
DECL FDAT Fl226={TOOL_NO 2,BASE_NO 3,IPO_FRAME #BASE,POINT2[] " "}
DECL E6POS Xl231={X 2212.30493,Y 49.1511192,Z 487.344086,A -102.423401,B 69.3434906,C 77.9126663,S 2,T 9,E1 0.0,E2 0.0,E3 0.0,E4 0.0,E5 0.0,E6 0.0}
DECL FDAT Fl231={TOOL_NO 2,BASE_NO 3,IPO_FRAME #BASE,POINT2[] " "}
DECL E6POS Xl236={X 2211.86694,Y 54.1603699,Z 500.974792,A -90.194397,B 69.8205338,C 89.3786697,S 2,T 9,E1 0.0,E2 0.0,E3 0.0,E4 0.0,E5 0.0,E6 0.0}
DECL FDAT Fl236={TOOL_NO 2,BASE_NO 3,IPO_FRAME #BASE,POINT2[] " ",TQ_STATE FALSE}
DECL E6POS Xl241={X 2186.20996,Y 60.8708115,Z 519.807617,A -90.1945267,B 69.820488,C 89.3785172,S 2,T 9,E1 0.0,E2 0.0,E3 0.0,E4 0.0,E5 0.0,E6 0.0}
DECL FDAT Fl241={TOOL_NO 2,BASE_NO 3,IPO_FRAME #BASE,POINT2[] " "}
DECL E6POS Xl242={X 2059.80493,Y 38.6424103,Z 487.18869,A -86.8489532,B 73.3499298,C 91.8619003,S 2,T 9,E1 0.0,E2 0.0,E3 0.0,E4 0.0,E5 0.0,E6 0.0}
DECL FDAT Fl242={TOOL_NO 2,BASE_NO 3,IPO_FRAME #BASE,POINT2[] " "}
DECL E6POS Xl246={X 2060.521,Y -63.3510208,Z 499.487793,A 100.750504,B 75.8574982,C -78.7533188,S 2,T 40,E1 0.0,E2 0.0,E3 0.0,E4 0.0,E5 0.0,E6 0.0}
DECL FDAT Fl246={TOOL_NO 2,BASE_NO 3,IPO_FRAME #BASE,POINT2[] " "}
DECL E6POS Xl251={X 2205.69702,Y -77.1784363,Z 511.767212,A 93.5408401,B 69.9691162,C -86.0749969,S 2,T 40,E1 0.0,E2 0.0,E3 0.0,E4 0.0,E5 0.0,E6 0.0}
DECL FDAT Fl251={TOOL_NO 2,BASE_NO 3,IPO_FRAME #BASE,POINT2[] " "}
DECL E6POS Xl256={X 2213.73901,Y -69.5282364,Z 490.48999,A 93.5408401,B 69.9691162,C -86.0749969,S 2,T 40,E1 0.0,E2 0.0,E3 0.0,E4 0.0,E5 0.0,E6 0.0}
DECL FDAT Fl256={TOOL_NO 2,BASE_NO 3,IPO_FRAME #BASE,POINT2[] " "}
DECL E6POS Xl261={X 2211.23511,Y -72.2856216,Z 498.151489,A 89.3737411,B 70.0178909,C -89.9905396,S 2,T 40,E1 0.0,E2 0.0,E3 0.0,E4 0.0,E5 0.0,E6 0.0}
DECL FDAT Fl261={TOOL_NO 2,BASE_NO 3,IPO_FRAME #BASE,POINT2[] " ",TQ_STATE FALSE}
DECL E6POS Xl262={X 2206.16089,Y -158.784607,Z 510.061401,A 70.9925919,B 78.4367523,C -110.064003,S 2,T 8,E1 0.0,E2 0.0,E3 0.0,E4 0.0,E5 0.0,E6 0.0}
DECL FDAT Fl262={TOOL_NO 2,BASE_NO 3,IPO_FRAME #BASE,POINT2[] " ",TQ_STATE FALSE}
DECL E6POS Xl266={X 2209.78101,Y -350.038513,Z 485.504913,A 89.4249573,B 88.7149429,C -90.5898132,S 2,T 8,E1 0.0,E2 0.0,E3 0.0,E4 0.0,E5 0.0,E6 0.0}
DECL FDAT Fl266={TOOL_NO 2,BASE_NO 3,IPO_FRAME #BASE,POINT2[] " "}
DECL E6POS Xl271={X 2207.95508,Y -402.089508,Z 465.060089,A -162.022797,B 86.4794617,C 18.0451107,S 2,T 8,E1 0.0,E2 0.0,E3 0.0,E4 0.0,E5 0.0,E6 0.0}
DECL FDAT Fl271={TOOL_NO 2,BASE_NO 3,IPO_FRAME #BASE,POINT2[] " ",TQ_STATE FALSE}
DECL LDAT LL_OLP80={VEL 1.0,ACC 100.0,APO_DIST 5.0,APO_FAC 0.0,ORI_TYP #VAR,CIRC_TYP #BASE,JERK_FAC 50.0}
DECL E6POS Xl276={X 2206.43506,Y -697.977417,Z 307.695404,A -97.4447174,B 75.2465363,C 82.46064,S 2,T 8,E1 0.0,E2 0.0,E3 0.0,E4 0.0,E5 0.0,E6 0.0}
DECL FDAT Fl276={TOOL_NO 2,BASE_NO 3,IPO_FRAME #BASE,POINT2[] " ",TQ_STATE FALSE}
DECL LDAT LL_OLP81={VEL 1.0,ACC 100.0,APO_DIST 5.0,APO_FAC 0.0,ORI_TYP #VAR,CIRC_TYP #BASE,JERK_FAC 50.0}
DECL E6POS Xl281={X 2205.229,Y -921.711975,Z 294.875,A -90.0,B 50.0000992,C 90.0,S 2,T 8}
DECL FDAT Fl281={TOOL_NO 2,BASE_NO 3,IPO_FRAME #BASE,POINT2[] " ",TQ_STATE FALSE}
DECL E6POS Xl286={X 2205.26904,Y -951.011414,Z 283.177307,A -90.0000916,B 50.0001907,C 89.9999619,S 2,T 8,E1 0.0,E2 0.0,E3 0.0,E4 0.0,E5 0.0,E6 0.0}
DECL FDAT Fl286={TOOL_NO 2,BASE_NO 3,IPO_FRAME #BASE,POINT2[] " ",TQ_STATE FALSE}
DECL E6POS Xl291={X 2210.24194,Y -936.010193,Z 302.306213,A -83.1879501,B 49.8001099,C 95.2132568,S 2,T 8,E1 0.0,E2 0.0,E3 0.0,E4 0.0,E5 0.0,E6 0.0}
DECL FDAT Fl291={TOOL_NO 2,BASE_NO 3,IPO_FRAME #BASE,POINT2[] " "}
DECL E6POS Xl296={X 2150.30005,Y -916.025818,Z 317.780914,A -89.9999924,B 50.0000992,C 90.0,S 2,T 8,E1 0.0,E2 0.0,E3 0.0,E4 0.0,E5 0.0,E6 0.0}
DECL FDAT Fl296={TOOL_NO 2,BASE_NO 3,IPO_FRAME #BASE,POINT2[] " "}
DECL PDAT PP_OLP37={VEL 100.0,ACC 100.0,APO_DIST 20.0,APO_MODE #CDIS}
DECL E6POS Xl301={X 1430.44604,Y -920.910889,Z 380.340912,A -65.894989,B 63.2542114,C -157.304199,S 2,T 9,E1 0.0,E2 0.0,E3 0.0,E4 0.0,E5 0.0,E6 0.0}
DECL FDAT Fl301={TOOL_NO 2,BASE_NO 3,IPO_FRAME #BASE,POINT2[] " ",TQ_STATE FALSE}
DECL LDAT LCPDAT0={VEL 2.0,ACC 100.0,APO_DIST 2.0,APO_FAC 50.0,AXIS_VEL 100.0,AXIS_ACC 100.0,ORI_TYP #VAR,CIRC_TYP #BASE,JERK_FAC 50.0,GEAR_JERK 50.0,EXAX_IGN 0}
DECL E6POS Xl306={X 1430.46106,Y -1010.914,Z 364.696106,A -66.584137,B 62.4910698,C -157.917603,S 2,T 9,E1 0.0,E2 0.0,E3 0.0,E4 0.0,E5 0.0,E6 0.0}
DECL FDAT Fl306={TOOL_NO 2,BASE_NO 3,IPO_FRAME #BASE,POINT2[] " "}
DECL LDAT LL_OLP85={VEL 1.0,ACC 100.0,APO_DIST 2.0,APO_FAC 0.0,ORI_TYP #VAR,CIRC_TYP #BASE,JERK_FAC 50.0}
DECL E6POS Xl311={X 1504.45801,Y -1015.81799,Z 309.69101,A -6.11479998,B 59.6772995,C -97.5519028,S 2,T 40}
DECL FDAT Fl311={TOOL_NO 2,BASE_NO 3,IPO_FRAME #BASE,POINT2[] " ",TQ_STATE FALSE}
DECL LDAT LL_OLP86={VEL 1.0,ACC 100.0,APO_DIST 5.0,APO_FAC 0.0,ORI_TYP #VAR,CIRC_TYP #BASE,JERK_FAC 50.0}
DECL E6POS Xl326={X 1408.64404,Y -1022.89801,Z 347.390106,A -119.316399,B 72.0361023,C 145.7341,S 2,T 8,E1 0.0,E2 0.0,E3 0.0,E4 0.0,E5 0.0,E6 0.0}
DECL FDAT Fl326={TOOL_NO 2,BASE_NO 3,IPO_FRAME #BASE,POINT2[] " ",TQ_STATE FALSE}
DECL LDAT LL_OLP87={VEL 1.0,ACC 100.0,APO_DIST 5.0,APO_FAC 0.0,ORI_TYP #VAR,CIRC_TYP #BASE,JERK_FAC 50.0}
DECL E6POS Xl331={X 1430.49805,Y -1010.927,Z 364.586212,A -69.6234894,B 58.5407104,C -160.565796,S 2,T 9,E1 0.0,E2 0.0,E3 0.0,E4 0.0,E5 0.0,E6 0.0}
DECL FDAT Fl331={TOOL_NO 2,BASE_NO 3,IPO_FRAME #BASE,POINT2[] " "}
DECL LDAT LL_OLP91={VEL 1.0,ACC 100.0,APO_DIST 20.0,APO_FAC 0.0,ORI_TYP #VAR,CIRC_TYP #BASE,JERK_FAC 50.0}
DECL E6POS Xl336={X 1430.45801,Y -920.916016,Z 371.963013,A -41.7638016,B 75.9057007,C -134.514694,S 2,T 40}
DECL FDAT Fl336={TOOL_NO 2,BASE_NO 3,IPO_FRAME #BASE,POINT2[] " "}
DECL E6POS Xl341={X 1023.37201,Y 195.498001,Z 1177.24402,A -56.0586014,B 67.5304031,C -3.93070006,S 2,T 10}
DECL FDAT Fl341={TOOL_NO 2,BASE_NO 3,IPO_FRAME #BASE,POINT2[] " ",TQ_STATE FALSE}
DECL E6POS Xl346={X 1231.26501,Y -831.768921,Z 1504.36499,A -95.0813599,B 7.10645723,C 1.27910495,S 6,T 27,E1 0.0,E2 0.0,E3 0.0,E4 0.0,E5 0.0,E6 0.0}
DECL FDAT Fl346={TOOL_NO 2,BASE_NO 3,IPO_FRAME #BASE,POINT2[] " "}
DECL E6POS Xl351={X 1236.73706,Y -925.240417,Z 1501.59998,A -95.1430511,B 4.8415041,C 1.23792803,S 6,T 27,E1 0.0,E2 0.0,E3 0.0,E4 0.0,E5 0.0,E6 0.0}
DECL FDAT Fl351={TOOL_NO 2,BASE_NO 3,IPO_FRAME #BASE,POINT2[] " "}
DECL LDAT LL_OLP92={VEL 1.0,ACC 100.0,APO_DIST 5.0,APO_FAC 0.0,ORI_TYP #VAR,CIRC_TYP #BASE,JERK_FAC 50.0}
DECL E6POS Xl327={X 1408.64404,Y -1022.89801,Z 347.390106,A -119.316399,B 72.0361023,C 145.7341,S 2,T 8,E1 0.0,E2 0.0,E3 0.0,E4 0.0,E5 0.0,E6 0.0}
DECL FDAT Fl327={TOOL_NO 2,BASE_NO 3,IPO_FRAME #BASE,POINT2[] " ",TQ_STATE FALSE}
DECL LDAT LL_OLP113={VEL 1.0,ACC 100.0,APO_DIST 5.0,APO_FAC 0.0,ORI_TYP #VAR,CIRC_TYP #BASE,JERK_FAC 50.0}
DECL E6POS Xl332={X 1430.49805,Y -1010.927,Z 364.586212,A -69.6234894,B 58.5407104,C -160.565796,S 2,T 9,E1 0.0,E2 0.0,E3 0.0,E4 0.0,E5 0.0,E6 0.0}
DECL FDAT Fl332={TOOL_NO 2,BASE_NO 3,IPO_FRAME #BASE,POINT2[] " "}
DECL LDAT LL_OLP114={VEL 1.0,ACC 100.0,APO_DIST 20.0,APO_FAC 0.0,ORI_TYP #VAR,CIRC_TYP #BASE,JERK_FAC 50.0}
DECL E6POS Xl337={X 1430.45801,Y -920.916016,Z 371.963013,A -41.7638016,B 75.9057007,C -134.514694,S 2,T 40}
DECL FDAT Fl337={TOOL_NO 2,BASE_NO 3,IPO_FRAME #BASE,POINT2[] " "}
DECL E6POS Xl342={X 1023.37201,Y 195.498001,Z 1177.24402,A -56.0586014,B 67.5304031,C -3.93070006,S 2,T 10}
DECL FDAT Fl342={TOOL_NO 2,BASE_NO 3,IPO_FRAME #BASE,POINT2[] " ",TQ_STATE FALSE}
DECL E6POS Xl347={X 1231.26501,Y -831.768921,Z 1504.36499,A -95.0813599,B 7.10645723,C 1.27910495,S 6,T 27,E1 0.0,E2 0.0,E3 0.0,E4 0.0,E5 0.0,E6 0.0}
DECL FDAT Fl347={TOOL_NO 2,BASE_NO 3,IPO_FRAME #BASE,POINT2[] " "}
DECL E6POS Xl352={X 1236.73706,Y -925.240417,Z 1501.59998,A -95.1430511,B 4.8415041,C 1.23792803,S 6,T 27,E1 0.0,E2 0.0,E3 0.0,E4 0.0,E5 0.0,E6 0.0}
DECL FDAT Fl352={TOOL_NO 2,BASE_NO 3,IPO_FRAME #BASE,POINT2[] " "}
DECL E6POS Xl356={X 1237.35205,Y -902.103821,Z 1502.85205,A -95.0070572,B 4.77904892,C 1.24916399,S 6,T 27,E1 0.0,E2 0.0,E3 0.0,E4 0.0,E5 0.0,E6 0.0}
DECL FDAT Fl356={TOOL_NO 2,BASE_NO 3,IPO_FRAME #BASE,POINT2[] " ",TQ_STATE FALSE}
DECL E6POS Xl366={X 1170.54395,Y -888.906677,Z 1500.99304,A -100.678802,B 6.10900593,C 0.468423009,S 6,T 27,E1 0.0,E2 0.0,E3 0.0,E4 0.0,E5 0.0,E6 0.0}
DECL FDAT Fl366={TOOL_NO 2,BASE_NO 3,IPO_FRAME #BASE,POINT2[] " ",TQ_STATE FALSE}
DECL E6POS Xl371={X 1072.00195,Y -914.824524,Z 1488.00598,A -109.049599,B 8.29882336,C -0.272952288,S 6,T 27,E1 0.0,E2 0.0,E3 0.0,E4 0.0,E5 0.0,E6 0.0}
DECL FDAT Fl371={TOOL_NO 2,BASE_NO 3,IPO_FRAME #BASE,POINT2[] " "}
DECL E6POS Xl376={X 1064.09204,Y -861.5896,Z 1491.30298,A -109.336899,B 8.1246233,C -0.28049019,S 6,T 27,E1 0.0,E2 0.0,E3 0.0,E4 0.0,E5 0.0,E6 0.0}
DECL FDAT Fl376={TOOL_NO 2,BASE_NO 3,IPO_FRAME #BASE,POINT2[] " ",TQ_STATE FALSE}
DECL E6POS Xl381={X 931.553711,Y -841.5177,Z 1564.98804,A -105.1548,B 6.91587019,C -3.35212302,S 6,T 27,E1 0.0,E2 0.0,E3 0.0,E4 0.0,E5 0.0,E6 0.0}
DECL FDAT Fl381={TOOL_NO 2,BASE_NO 3,IPO_FRAME #BASE,POINT2[] " "}
DECL E6POS Xl421={X 764.0047,Y -856.662781,Z 1555.68201,A -106.300598,B 8.76704121,C 1.16544497,S 6,T 59,E1 0.0,E2 0.0,E3 0.0,E4 0.0,E5 0.0,E6 0.0}
DECL FDAT Fl421={TOOL_NO 2,BASE_NO 3,IPO_FRAME #BASE,POINT2[] " "}
DECL E6POS Xl431={X 662.682617,Y -894.061279,Z 1477.90198,A -111.868599,B 12.2453203,C 1.99518895,S 6,T 58,E1 0.0,E2 0.0,E3 0.0,E4 0.0,E5 0.0,E6 0.0}
DECL FDAT Fl431={TOOL_NO 2,BASE_NO 3,IPO_FRAME #BASE,POINT2[] " "}
DECL E6POS Xl436={X 668.38031,Y -879.865479,Z 1481.22205,A -111.868599,B 12.2453203,C 1.99518895,S 6,T 59,E1 0.0,E2 0.0,E3 0.0,E4 0.0,E5 0.0,E6 0.0}
DECL FDAT Fl436={TOOL_NO 2,BASE_NO 3,IPO_FRAME #BASE,POINT2[] " ",TQ_STATE FALSE}
DECL E6POS Xl441={X 903.630981,Y -565.390015,Z 1544.61304,A -115.101402,B 14.6844997,C 2.03340006,S 6,T 27,E1 0.0,E2 0.0,E3 0.0,E4 0.0,E5 0.0,E6 0.0}
DECL FDAT Fl441={TOOL_NO 2,BASE_NO 3,IPO_FRAME #BASE,POINT2[] " "}
DECL PDAT PP_OLP46={VEL 100.0,ACC 100.0,APO_DIST 50.0,APO_MODE #CDIS}
DECL E6POS Xl451={X 1399.95703,Y -542.234924,Z 2580.37402,A -75.9914017,B 22.5326004,C -25.0158005,S 6,T 27,E1 0.0,E2 0.0,E3 0.0,E4 0.0,E5 0.0,E6 0.0}
DECL FDAT Fl451={TOOL_NO 2,BASE_NO 3,IPO_FRAME #BASE,POINT2[] " ",TQ_STATE FALSE}
DECL PDAT PPDAT40={VEL 100.0,ACC 100.0,APO_DIST 50.0,APO_MODE #CDIS}
DECL E6POS XP3={X 2558.93188,Y -485.116211,Z 3441.69092,A -36.1692314,B -13.5166597,C 1.14306998,S 6,T 27,E1 0.0,E2 0.0,E3 0.0,E4 0.0,E5 0.0,E6 0.0}
DECL FDAT FP3={TOOL_NO 2,BASE_NO 3,IPO_FRAME #BASE,POINT2[] " ",TQ_STATE FALSE}
DECL PDAT PPDAT41={VEL 100.0,ACC 100.0,APO_DIST 50.0,APO_MODE #CDIS}
DECL E6POS XP4={X 2641.70508,Y 753.610291,Z 4294.20215,A 42.6114388,B -30.1368103,C -35.3248711,S 2,T 11,E1 0.0,E2 0.0,E3 0.0,E4 0.0,E5 0.0,E6 0.0}
DECL FDAT FP4={TOOL_NO 2,BASE_NO 3,IPO_FRAME #BASE,POINT2[] " ",TQ_STATE FALSE}
DECL PDAT PPDAT42={VEL 100.0,ACC 100.0,APO_DIST 50.0,APO_MODE #CDIS}
DECL E6POS XP5={X 1807.78699,Y 389.460297,Z 3419.56201,A 63.818779,B 37.8043785,C -38.9489098,S 2,T 2,E1 0.0,E2 0.0,E3 0.0,E4 0.0,E5 0.0,E6 0.0}
DECL FDAT FP5={TOOL_NO 2,BASE_NO 3,IPO_FRAME #BASE,POINT2[] " ",TQ_STATE FALSE}
DECL PDAT PP_OLP50={VEL 100.0,ACC 100.0,APO_DIST 50.0,APO_MODE #CDIS}
DECL E6POS Xl032={X 1052.75195,Y 58.7190018,Z 2073.41504,A -29.1716995,B 74.7963028,C -24.9258003,S 2,T 3}
DECL FDAT Fl032={TOOL_NO 2,BASE_NO 3,IPO_FRAME #BASE,POINT2[] " ",TQ_STATE FALSE}
DECL E6POS Xl232={X 2212.302,Y 51.1460686,Z 487.354187,A -97.8317184,B 69.6583862,C 82.8152771,S 2,T 9,E1 0.0,E2 0.0,E3 0.0,E4 0.0,E5 0.0,E6 0.0}
DECL FDAT Fl232={TOOL_NO 2,BASE_NO 3,IPO_FRAME #BASE,POINT2[] " "}
DECL E6POS Xl446={X 1399.11096,Y -542.002991,Z 2358.92798,A -75.9914017,B 22.5326004,C -25.0158005,S 2,T 11}
DECL FDAT Fl446={TOOL_NO 2,BASE_NO 3,IPO_FRAME #BASE,POINT2[] " ",TQ_STATE FALSE}
DECL E6POS XP6={X 1581.85901,Y 261.861115,Z 2436.37891,A 32.6823807,B 53.7033081,C 6.08660078,S 2,T 3,E1 0.0,E2 0.0,E3 0.0,E4 0.0,E5 0.0,E6 0.0}
DECL FDAT FP6={TOOL_NO 2,BASE_NO 3,IPO_FRAME #BASE,POINT2[] " ",TQ_STATE FALSE}
DECL E6POS Xl035={X 1052.75195,Y 58.7190018,Z 2073.41504,A -29.1716995,B 74.7963028,C -24.9258003}
DECL FDAT Fl035={TOOL_NO 2,BASE_NO 3,IPO_FRAME #BASE,POINT2[] " ",TQ_STATE FALSE}
DECL E6POS Xl037={X 865.1698,Y -552.292908,Z 1653.08899,A 72.2369766,B 83.6307907,C 36.7096405,S 2,T 2,E1 0.0,E2 0.0,E3 0.0,E4 0.0,E5 0.0,E6 0.0}
DECL FDAT Fl037={TOOL_NO 2,BASE_NO 3,IPO_FRAME #BASE,POINT2[] " "}
DECL E6POS Xl416={X 672.293518,Y -882.395874,Z 1477.16699,A -112.8713,B 9.92592716,C -1.17351198,S 2,T 11,E1 0.0,E2 0.0,E3 0.0,E4 0.0,E5 0.0,E6 0.0}
DECL FDAT Fl416={TOOL_NO 2,BASE_NO 3,IPO_FRAME #BASE,POINT2[] " "}
DECL E6POS Xl437={X 745.929688,Y -761.459106,Z 1505.35498,A -118.336403,B 11.7002602,C 1.16059995,S 2,T 11,E1 0.0,E2 0.0,E3 0.0,E4 0.0,E5 0.0,E6 0.0}
DECL FDAT Fl437={TOOL_NO 2,BASE_NO 3,IPO_FRAME #BASE,POINT2[] " "}
DECL E6POS Xl442={X 903.630981,Y -565.390015,Z 1544.61304,A -115.101402,B 14.6844997,C 2.03340006,S 2,T 11}
DECL FDAT Fl442={TOOL_NO 2,BASE_NO 3,IPO_FRAME #BASE,POINT2[] " ",TQ_STATE FALSE}
DECL PDAT PPDAT43={VEL 100.0,ACC 100.0,APO_DIST 50.0,APO_MODE #CDIS}
DECL E6POS XP7={X 1163.45496,Y -648.34668,Z 1812.50806,A -102.584297,B 11.4974098,C -2.25978899,S 2,T 11,E1 0.0,E2 0.0,E3 0.0,E4 0.0,E5 0.0,E6 0.0}
DECL FDAT FP7={TOOL_NO 2,BASE_NO 3,IPO_FRAME #BASE,POINT2[] " ",TQ_STATE FALSE}
DECL E6POS Xl417={X 672.293518,Y -882.395874,Z 1477.16699,A -112.8713,B 9.92592716,C -1.17351198,S 2,T 11,E1 0.0,E2 0.0,E3 0.0,E4 0.0,E5 0.0,E6 0.0}
DECL FDAT Fl417={TOOL_NO 2,BASE_NO 3,IPO_FRAME #BASE,POINT2[] " "}
DECL E6POS Xl438={X 745.929688,Y -761.459106,Z 1505.35498,A -118.336403,B 11.7002602,C 1.16059995,S 2,T 11,E1 0.0,E2 0.0,E3 0.0,E4 0.0,E5 0.0,E6 0.0}
DECL FDAT Fl438={TOOL_NO 2,BASE_NO 3,IPO_FRAME #BASE,POINT2[] " "}
DECL E6POS Xl443={X 903.630981,Y -565.390015,Z 1544.61304,A -115.101402,B 14.6844997,C 2.03340006,S 2,T 11}
DECL FDAT Fl443={TOOL_NO 2,BASE_NO 3,IPO_FRAME #BASE,POINT2[] " ",TQ_STATE FALSE}
DECL PDAT PPDAT44={VEL 100.0,ACC 100.0,APO_DIST 50.0,APO_MODE #CDIS}
DECL E6POS XP8={X 1163.45496,Y -648.34668,Z 1812.50806,A -102.584297,B 11.4974098,C -2.25978899,S 2,T 11,E1 0.0,E2 0.0,E3 0.0,E4 0.0,E5 0.0,E6 0.0}
DECL FDAT FP8={TOOL_NO 2,BASE_NO 3,IPO_FRAME #BASE,POINT2[] " ",TQ_STATE FALSE}
DECL E6POS Xl439={X 668.38031,Y -879.865479,Z 1481.22205,A -111.868599,B 12.2453203,C 1.99518895,S 6,T 59,E1 0.0,E2 0.0,E3 0.0,E4 0.0,E5 0.0,E6 0.0}
DECL FDAT Fl439={TOOL_NO 2,BASE_NO 3,IPO_FRAME #BASE,POINT2[] " ",TQ_STATE FALSE}
DECL E6POS Xl444={X 903.630981,Y -565.390015,Z 1544.61304,A -115.101402,B 14.6844997,C 2.03340006,S 6,T 27,E1 0.0,E2 0.0,E3 0.0,E4 0.0,E5 0.0,E6 0.0}
DECL FDAT Fl444={TOOL_NO 2,BASE_NO 3,IPO_FRAME #BASE,POINT2[] " "}
DECL PDAT PP_OLP51={VEL 100.0,ACC 100.0,APO_DIST 50.0,APO_MODE #CDIS}
DECL E6POS Xl452={X 1399.95703,Y -542.234924,Z 2580.37402,A -75.9914017,B 22.5326004,C -25.0158005,S 6,T 27,E1 0.0,E2 0.0,E3 0.0,E4 0.0,E5 0.0,E6 0.0}
DECL FDAT Fl452={TOOL_NO 2,BASE_NO 3,IPO_FRAME #BASE,POINT2[] " ",TQ_STATE FALSE}
DECL PDAT PPDAT45={VEL 100.0,ACC 100.0,APO_DIST 50.0,APO_MODE #CDIS}
DECL E6POS XP9={X 2558.93188,Y -485.116211,Z 3441.69092,A -36.1692314,B -13.5166597,C 1.14306998,S 6,T 27,E1 0.0,E2 0.0,E3 0.0,E4 0.0,E5 0.0,E6 0.0}
DECL FDAT FP9={TOOL_NO 2,BASE_NO 3,IPO_FRAME #BASE,POINT2[] " ",TQ_STATE FALSE}
DECL PDAT PPDAT46={VEL 100.0,ACC 100.0,APO_DIST 50.0,APO_MODE #CDIS}
DECL E6POS XP10={X 2641.70508,Y 753.610291,Z 4294.20215,A 42.6114388,B -30.1368103,C -35.3248711,S 2,T 11,E1 0.0,E2 0.0,E3 0.0,E4 0.0,E5 0.0,E6 0.0}
DECL FDAT FP10={TOOL_NO 2,BASE_NO 3,IPO_FRAME #BASE,POINT2[] " ",TQ_STATE FALSE}
DECL PDAT PPDAT47={VEL 100.0,ACC 100.0,APO_DIST 50.0,APO_MODE #CDIS}
DECL E6POS XP11={X 1544.94702,Y 683.336914,Z 2350.90894,A 40.8428001,B 47.0746803,C 31.0701103,S 2,T 11,E1 0.0,E2 0.0,E3 0.0,E4 0.0,E5 0.0,E6 0.0}
DECL FDAT FP11={TOOL_NO 2,BASE_NO 3,IPO_FRAME #BASE,POINT2[] " ",TQ_STATE FALSE}
DECL PDAT PP_OLP52={VEL 100.0,ACC 100.0,APO_DIST 50.0,APO_MODE #CDIS}
DECL E6POS Xl040={X 1052.75195,Y 58.7190018,Z 2073.41504,A -29.1716995,B 74.7963028,C -24.9258003,S 2,T 3}
DECL FDAT Fl040={TOOL_NO 2,BASE_NO 3,IPO_FRAME #BASE,POINT2[] " ",TQ_STATE FALSE}
DECL E6POS XP12={X 331.4263,Y -869.018982,Z -1.62679398,A 168.843704,B 71.7335968,C 101.289497,S 2,T 0,E1 0.0,E2 0.0,E3 0.0,E4 0.0,E5 0.0,E6 0.0}
DECL FDAT FP12={TOOL_NO 2,BASE_NO 3,IPO_FRAME #BASE,POINT2[] " ",TQ_STATE FALSE}
DECL E6POS Xl144={X 274.793304,Y -976.535583,Z -18.3775806,A -155.126495,B 79.2150497,C 141.135803,S 2,T 0,E1 0.0,E2 0.0,E3 0.0,E4 0.0,E5 0.0,E6 0.0}
DECL FDAT Fl144={TOOL_NO 2,BASE_NO 3,IPO_FRAME #BASE,POINT2[] " ",TQ_STATE FALSE}
DECL E6POS Xl149={X 271.043213,Y -986.491699,Z -31.1311302,A 177.039307,B 81.2389374,C 113.696999,S 2,T 0,E1 0.0,E2 0.0,E3 0.0,E4 0.0,E5 0.0,E6 0.0}
DECL FDAT Fl149={TOOL_NO 2,BASE_NO 3,IPO_FRAME #BASE,POINT2[] " "}
DECL LDAT LCPDAT29={VEL 2.0,ACC 100.0,APO_DIST 100.0,APO_FAC 50.0,AXIS_VEL 100.0,AXIS_ACC 100.0,ORI_TYP #VAR,CIRC_TYP #BASE,JERK_FAC 50.0,GEAR_JERK 50.0,EXAX_IGN 0}
DECL E6POS XSWP_60_7099={X 282.618805,Y -978.388123,Z -47.8770103,A 137.079605,B 82.4564972,C 73.1910477,S 2,T 0,E1 0.0,E2 0.0,E3 0.0,E4 0.0,E5 0.0,E6 0.0}
DECL FDAT FSWP_60_7099={TOOL_NO 2,BASE_NO 3,IPO_FRAME #BASE,POINT2[] " ",TQ_STATE FALSE}
DECL LDAT LL_OLP144={VEL 2.0,ACC 100.0,APO_DIST 0.0,APO_FAC 0.0,ORI_TYP #VAR,CIRC_TYP #BASE,JERK_FAC 50.0}
DECL E6POS XSWP_60_7100={X 228.0858,Y 955.865906,Z -30.4408398,A -158.172806,B 60.0438118,C -90.2183228,S 2,T 41,E1 0.0,E2 0.0,E3 0.0,E4 0.0,E5 0.0,E6 0.0}
DECL FDAT FSWP_60_7100={TOOL_NO 2,BASE_NO 3,IPO_FRAME #BASE,POINT2[] " ",TQ_STATE FALSE}
DECL LDAT LL_OLP145={VEL 2.0,ACC 100.0,APO_DIST 0.0,APO_FAC 0.0,ORI_TYP #VAR,CIRC_TYP #BASE,JERK_FAC 50.0}
DECL E6POS XSWP_60_7101={X 257.398987,Y 968.362793,Z -36.2217598,A -159.207306,B 74.111557,C -91.3095932,S 2,T 9,E1 0.0,E2 0.0,E3 0.0,E4 0.0,E5 0.0,E6 0.0}
DECL FDAT FSWP_60_7101={TOOL_NO 2,BASE_NO 3,IPO_FRAME #BASE,POINT2[] " ",TQ_STATE FALSE}
DECL LDAT LL_OLP146={VEL 1.0,ACC 100.0,APO_DIST 50.0,APO_FAC 0.0,ORI_TYP #VAR,CIRC_TYP #BASE,JERK_FAC 50.0}
DECL E6POS Xl042={X 267.976501,Y 976.090088,Z -36.6190109,A -159.346802,B 77.9462128,C -92.8242264,S 2,T 9,E1 0.0,E2 0.0,E3 0.0,E4 0.0,E5 0.0,E6 0.0}
DECL FDAT Fl042={TOOL_NO 9,BASE_NO 3,IPO_FRAME #BASE,POINT2[] " "}
DECL LDAT LL_OLP147={VEL 2.0,ACC 100.0,APO_DIST 0.0,APO_FAC 0.0,ORI_TYP #VAR,CIRC_TYP #BASE,JERK_FAC 50.0}
DECL E6POS XSWP_60_7102={X 285.441803,Y 980.617126,Z -43.8651619,A -157.531998,B 82.9950027,C -93.2139969,S 2,T 9,E1 0.0,E2 0.0,E3 0.0,E4 0.0,E5 0.0,E6 0.0}
DECL FDAT FSWP_60_7102={TOOL_NO 2,BASE_NO 3,IPO_FRAME #BASE,POINT2[] " ",TQ_STATE FALSE}
DECL E6POS Xl045={X 278.522888,Y 984.941711,Z -37.2186317,A 162.097397,B 82.7963715,C -133.723404,S 2,T 9,E1 0.0,E2 0.0,E3 0.0,E4 0.0,E5 0.0,E6 0.0}
DECL FDAT Fl045={TOOL_NO 2,BASE_NO 3,IPO_FRAME #BASE,POINT2[] " ",TQ_STATE FALSE}
DECL E6POS Xl047={X 256.019989,Y 971.379089,Z -11.6124401,A -179.4879,B 63.4032211,C -98.589241,S 2,T 41,E1 0.0,E2 0.0,E3 0.0,E4 0.0,E5 0.0,E6 0.0}
DECL FDAT Fl047={TOOL_NO 2,BASE_NO 3,IPO_FRAME #BASE,POINT2[] " "}
DECL E6POS Xl050={X 293.173004,Y 908.471985,Z -4.25699997,A -179.468597,B 64.332901,C -98.5838013,S 2,T 41}
DECL FDAT Fl050={TOOL_NO 2,BASE_NO 3,IPO_FRAME #BASE,POINT2[] " "}
DECL PDAT Pxxlarge={VEL 100.0,ACC 100.0,APO_DIST 1000.0,APO_MODE #CDIS}
DECL E6POS Xl053={X 685.003906,Y 846.773987,Z 261.842804,A 132.399994,B 71.1641312,C -138.405899,S 2,T 8,E1 0.0,E2 0.0,E3 0.0,E4 0.0,E5 0.0,E6 0.0}
DECL FDAT Fl053={TOOL_NO 2,BASE_NO 3,IPO_FRAME #BASE,POINT2[] " ",TQ_STATE FALSE}
DECL E6POS Xl088={X 982.077026,Y 804.691711,Z 1286.95996,A 130.202194,B 72.0134735,C -140.721497,S 2,T 10,E1 0.0,E2 0.0,E3 0.0,E4 0.0,E5 0.0,E6 0.0}
DECL FDAT Fl088={TOOL_NO 2,BASE_NO 3,IPO_FRAME #BASE,POINT2[] " "}
DECL E6POS Xl118={X 1264.32202,Y 229.841003,Z 1660.927,A 90.9709625,B 45.0197487,C -22.2856197,S 6,T 18,E1 0.0,E2 0.0,E3 0.0,E4 0.0,E5 0.0,E6 0.0}
DECL FDAT Fl118={TOOL_NO 2,BASE_NO 3,IPO_FRAME #BASE,POINT2[] " ",TQ_STATE FALSE}
DECL LDAT LL_OLP183={VEL 2.0,ACC 100.0,APO_DIST 0.0,APO_FAC 0.0,ORI_TYP #VAR,CIRC_TYP #BASE,JERK_FAC 50.0}
DECL E6POS XSWP_60_7103={X 257.140991,Y -965.624573,Z -42.9534607,A 147.275894,B 69.8397903,C 80.1007004,S 2,T 0,E1 0.0,E2 0.0,E3 0.0,E4 0.0,E5 0.0,E6 0.0}
DECL FDAT FSWP_60_7103={TOOL_NO 2,BASE_NO 3,IPO_FRAME #BASE,POINT2[] " ",TQ_STATE FALSE}
DECL LDAT LL_OLP185={VEL 2.0,ACC 100.0,APO_DIST 0.0,APO_FAC 0.0,ORI_TYP #VAR,CIRC_TYP #BASE,JERK_FAC 50.0}
DECL E6POS XSWP_60_7104={X 227.981903,Y -953.713501,Z -32.7617493,A 156.240295,B 60.0344696,C 88.5653229,S 2,T 0,E1 0.0,E2 0.0,E3 0.0,E4 0.0,E5 0.0,E6 0.0}
DECL FDAT FSWP_60_7104={TOOL_NO 2,BASE_NO 3,IPO_FRAME #BASE,POINT2[] " ",TQ_STATE FALSE}
DECL LDAT LL_OLP186={VEL 2.0,ACC 100.0,APO_DIST 0.0,APO_FAC 0.0,ORI_TYP #VAR,CIRC_TYP #BASE,JERK_FAC 50.0}
DECL E6POS XSWP_60_7105={X 221.412094,Y -949.96228,Z -9.63102055,A 159.264694,B 57.0288696,C 89.6700363,S 2,T 0,E1 0.0,E2 0.0,E3 0.0,E4 0.0,E5 0.0,E6 0.0}
DECL FDAT FSWP_60_7105={TOOL_NO 2,BASE_NO 3,IPO_FRAME #BASE,POINT2[] " ",TQ_STATE FALSE}
DECL E6POS Xl159={X 241.036804,Y -968.442627,Z -17.8401203,A 160.223801,B 57.3985481,C 89.056282,S 2,T 0,E1 0.0,E2 0.0,E3 0.0,E4 0.0,E5 0.0,E6 0.0}
DECL FDAT Fl159={TOOL_NO 2,BASE_NO 3,IPO_FRAME #BASE,POINT2[] " ",TQ_STATE FALSE}
DECL E6POS XP13={X 248.994797,Y -971.716675,Z -15.9355297,A 171.397003,B 59.5439415,C 94.138237,S 2,T 0,E1 0.0,E2 0.0,E3 0.0,E4 0.0,E5 0.0,E6 0.0}
DECL FDAT FP13={TOOL_NO 2,BASE_NO 3,IPO_FRAME #BASE,POINT2[] " ",TQ_STATE FALSE}
DECL E6POS Xl164={X 263.451294,Y -942.957886,Z -9.79736233,A 173.132294,B 58.8152618,C 94.1062927,S 2,T 0,E1 0.0,E2 0.0,E3 0.0,E4 0.0,E5 0.0,E6 0.0}
DECL FDAT Fl164={TOOL_NO 2,BASE_NO 3,IPO_FRAME #BASE,POINT2[] " "}
DECL E6POS Xl174={X 359.818787,Y -638.44342,Z 194.3862,A 153.228806,B 80.0036392,C 122.754997,S 2,T 0,E1 0.0,E2 0.0,E3 0.0,E4 0.0,E5 0.0,E6 0.0}
DECL FDAT Fl174={TOOL_NO 2,BASE_NO 3,IPO_FRAME #BASE,POINT2[] " ",TQ_STATE FALSE}
DECL E6POS Xl177={X 426.982208,Y -459.071503,Z 415.45639,A -124.0821,B 82.0942993,C -133.209793,S 2,T 0,E1 0.0,E2 0.0,E3 0.0,E4 0.0,E5 0.0,E6 0.0}
DECL FDAT Fl177={TOOL_NO 2,BASE_NO 3,IPO_FRAME #BASE,POINT2[] " ",TQ_STATE FALSE}
DECL PDAT PP_OLP92={VEL 100.0,ACC 100.0,APO_DIST 0.0}
DECL E6POS Xl178={X 653.832581,Y 465.707611,Z 389.711212,A 133.309494,B 81.4104538,C -175.386993,S 2,T 8,E1 0.0,E2 0.0,E3 0.0,E4 0.0,E5 0.0,E6 0.0}
DECL FDAT Fl178={TOOL_NO 2,BASE_NO 3,IPO_FRAME #BASE,POINT2[] " ",TQ_STATE FALSE}
DECL E6POS XP14={X 414.20929,Y 772.79718,Z 247.5634,A -175.614502,B 70.4779282,C -106.980904,S 2,T 9,E1 0.0,E2 0.0,E3 0.0,E4 0.0,E5 0.0,E6 0.0}
DECL FDAT FP14={TOOL_NO 2,BASE_NO 3,IPO_FRAME #BASE,POINT2[] " ",TQ_STATE FALSE}
DECL E6POS Xl051={X 293.173004,Y 908.471985,Z -4.25699997,A -179.468597,B 64.332901,C -98.5838013,S 2,T 41}
DECL FDAT Fl051={TOOL_NO 2,BASE_NO 3,IPO_FRAME #BASE,POINT2[] " ",TQ_STATE FALSE}
DECL E6POS Xl052={X 246.361694,Y 969.565918,Z -10.3455696,A -178.005005,B 59.3805008,C -97.2920685,S 2,T 41,E1 0.0,E2 0.0,E3 0.0,E4 0.0,E5 0.0,E6 0.0}
DECL FDAT Fl052={TOOL_NO 2,BASE_NO 3,IPO_FRAME #BASE,POINT2[] " "}
DECL E6POS Xl054={X 232.896103,Y 965.467102,Z -23.4360504,A -168.154404,B 59.6470985,C -98.7977982,S 2,T 41,E1 0.0,E2 0.0,E3 0.0,E4 0.0,E5 0.0,E6 0.0}
DECL FDAT Fl054={TOOL_NO 2,BASE_NO 3,IPO_FRAME #BASE,POINT2[] " "}
DECL LDAT LL_OLP143={VEL 2.0,ACC 100.0,APO_DIST 0.0,APO_FAC 0.0,ORI_TYP #VAR,CIRC_TYP #BASE,JERK_FAC 50.0}
DECL E6POS XSWP_60_7106={X 220.999802,Y 949.255188,Z -5.67109823,A -158.218002,B 60.0423508,C -90.2030563,S 2,T 41,E1 0.0,E2 0.0,E3 0.0,E4 0.0,E5 0.0,E6 0.0}
DECL FDAT FSWP_60_7106={TOOL_NO 2,BASE_NO 3,IPO_FRAME #BASE,POINT2[] " ",TQ_STATE FALSE}
DECL LDAT LL_OLP148={VEL 2.0,ACC 100.0,APO_DIST 0.0,APO_FAC 0.0,ORI_TYP #VAR,CIRC_TYP #BASE,JERK_FAC 50.0}
DECL E6POS XSWP_60_7107={X 228.0858,Y 955.865906,Z -30.4408398,A -158.172806,B 60.0438118,C -90.2183228,S 2,T 41,E1 0.0,E2 0.0,E3 0.0,E4 0.0,E5 0.0,E6 0.0}
DECL FDAT FSWP_60_7107={TOOL_NO 2,BASE_NO 3,IPO_FRAME #BASE,POINT2[] " ",TQ_STATE FALSE}
DECL LDAT LL_OLP149={VEL 2.0,ACC 100.0,APO_DIST 0.0,APO_FAC 0.0,ORI_TYP #VAR,CIRC_TYP #BASE,JERK_FAC 50.0}
DECL E6POS XSWP_60_7108={X 257.398987,Y 968.362793,Z -36.2217598,A -159.207306,B 74.111557,C -91.3095932,S 2,T 9,E1 0.0,E2 0.0,E3 0.0,E4 0.0,E5 0.0,E6 0.0}
DECL FDAT FSWP_60_7108={TOOL_NO 2,BASE_NO 3,IPO_FRAME #BASE,POINT2[] " ",TQ_STATE FALSE}
DECL LDAT LL_OLP150={VEL 1.0,ACC 100.0,APO_DIST 50.0,APO_FAC 0.0,ORI_TYP #VAR,CIRC_TYP #BASE,JERK_FAC 50.0}
DECL E6POS Xl055={X 267.976501,Y 976.090088,Z -36.6190109,A -159.346802,B 77.9462128,C -92.8242264,S 2,T 9,E1 0.0,E2 0.0,E3 0.0,E4 0.0,E5 0.0,E6 0.0}
DECL FDAT Fl055={TOOL_NO 9,BASE_NO 3,IPO_FRAME #BASE,POINT2[] " "}
DECL LDAT LL_OLP151={VEL 2.0,ACC 100.0,APO_DIST 0.0,APO_FAC 0.0,ORI_TYP #VAR,CIRC_TYP #BASE,JERK_FAC 50.0}
DECL E6POS XSWP_60_7109={X 285.441803,Y 980.617126,Z -43.8651619,A -157.531998,B 82.9950027,C -93.2139969,S 2,T 9,E1 0.0,E2 0.0,E3 0.0,E4 0.0,E5 0.0,E6 0.0}
DECL FDAT FSWP_60_7109={TOOL_NO 2,BASE_NO 3,IPO_FRAME #BASE,POINT2[] " ",TQ_STATE FALSE}
DECL E6POS Xl056={X 278.522888,Y 984.941711,Z -37.2186317,A 162.097397,B 82.7963715,C -133.723404,S 2,T 9,E1 0.0,E2 0.0,E3 0.0,E4 0.0,E5 0.0,E6 0.0}
DECL FDAT Fl056={TOOL_NO 2,BASE_NO 3,IPO_FRAME #BASE,POINT2[] " ",TQ_STATE FALSE}
DECL E6POS Xl057={X 256.019989,Y 971.379089,Z -11.6124401,A -179.4879,B 63.4032211,C -98.589241,S 2,T 41,E1 0.0,E2 0.0,E3 0.0,E4 0.0,E5 0.0,E6 0.0}
DECL FDAT Fl057={TOOL_NO 2,BASE_NO 3,IPO_FRAME #BASE,POINT2[] " "}
DECL E6POS Xl058={X 293.173004,Y 908.471985,Z -4.25699997,A -179.468597,B 64.332901,C -98.5838013,S 2,T 41}
DECL FDAT Fl058={TOOL_NO 2,BASE_NO 3,IPO_FRAME #BASE,POINT2[] " "}
DECL E6POS Xl059={X 685.003906,Y 846.773987,Z 261.842804,A 132.399994,B 71.1641312,C -138.405899,S 2,T 8,E1 0.0,E2 0.0,E3 0.0,E4 0.0,E5 0.0,E6 0.0}
DECL FDAT Fl059={TOOL_NO 2,BASE_NO 3,IPO_FRAME #BASE,POINT2[] " ",TQ_STATE FALSE}
DECL E6POS Xl089={X 982.077026,Y 804.691711,Z 1286.95996,A 130.202194,B 72.0134735,C -140.721497,S 2,T 10,E1 0.0,E2 0.0,E3 0.0,E4 0.0,E5 0.0,E6 0.0}
DECL FDAT Fl089={TOOL_NO 2,BASE_NO 3,IPO_FRAME #BASE,POINT2[] " "}
DECL E6POS Xl119={X 1264.32202,Y 229.841003,Z 1660.927,A 90.9709625,B 45.0197487,C -22.2856197,S 6,T 18,E1 0.0,E2 0.0,E3 0.0,E4 0.0,E5 0.0,E6 0.0}
DECL FDAT Fl119={TOOL_NO 2,BASE_NO 3,IPO_FRAME #BASE,POINT2[] " ",TQ_STATE FALSE}
DECL E6POS Xl179={X 1656.474,Y 70.8213577,Z 1898.63,A 85.0365067,B 50.6858101,C -24.4635792,S 2,T 2,E1 0.0,E2 0.0,E3 0.0,E4 0.0,E5 0.0,E6 0.0}
DECL FDAT Fl179={TOOL_NO 2,BASE_NO 3,IPO_FRAME #BASE,POINT2[] " ",TQ_STATE FALSE}
DECL PDAT PPDAT48={VEL 100.0,ACC 100.0,APO_DIST 50.0,APO_MODE #CDIS}
DECL E6POS XP15={X 1807.78406,Y 389.461395,Z 3419.56104,A 63.8191414,B 37.8045616,C -38.9490814,S 2,T 3,E1 0.0,E2 0.0,E3 0.0,E4 0.0,E5 0.0,E6 0.0}
DECL FDAT FP15={TOOL_NO 2,BASE_NO 3,IPO_FRAME #BASE,POINT2[] " ",TQ_STATE FALSE}
DECL E6POS Xl060={X 1110.92896,Y 490.82251,Z 1769.04504,A 121.191299,B 20.5780697,C -14.8572798,S 2,T 10,E1 0.0,E2 0.0,E3 0.0,E4 0.0,E5 0.0,E6 0.0}
DECL FDAT Fl060={TOOL_NO 2,BASE_NO 3,IPO_FRAME #BASE,POINT2[] " ",TQ_STATE FALSE}
DECL E6POS Xl061={X 1052.75195,Y 58.7190018,Z 2073.41504,A -29.1716995,B 74.7963028,C -24.9258003,S 2,T 3}
DECL FDAT Fl061={TOOL_NO 2,BASE_NO 3,IPO_FRAME #BASE,POINT2[] " ",TQ_STATE FALSE}
DECL PDAT PPDAT49={VEL 100.0,ACC 100.0,APO_DIST 50.0,APO_MODE #CDIS}
DECL E6POS XP16={X 764.261414,Y -310.796112,Z 1324.02295,A -118.439201,B 84.7641373,C -144.651398,S 2,T 3,E1 0.0,E2 0.0,E3 0.0,E4 0.0,E5 0.0,E6 0.0}
DECL FDAT FP16={TOOL_NO 2,BASE_NO 3,IPO_FRAME #BASE,POINT2[] " ",TQ_STATE FALSE}
ENDDAT
